C03637=1034.949,55.680,408.696,168.997,41.142,157.715
C03638=1034.955,55.929,408.679,168.999,41.142,157.715
C03639=1034.961,56.179,408.661,169.001,41.141,157.715
C03640=1034.968,56.428,408.644,169.004,41.140,157.715
C03641=1034.974,56.677,408.627,169.006,41.140,157.715
C03642=1034.980,56.927,408.610,169.008,41.139,157.715
C03643=1034.986,57.176,408.593,169.010,41.139,157.715
C03644=1034.993,57.425,408.576,169.012,41.139,157.715
C03645=1034.999,57.675,408.558,169.015,41.138,157.715
C03646=1035.006,57.924,408.541,169.017,41.138,157.715
C03647=1035.012,58.174,408.523,169.019,41.137,157.715
C03648=1035.018,58.423,408.505,169.021,41.136,157.715
C03649=1035.025,58.672,408.488,169.023,41.136,157.715
C03650=1035.031,58.921,408.470,169.026,41.136,157.715
C03651=1035.038,59.171,408.453,169.028,41.135,157.715
C03652=1035.044,59.420,408.436,169.030,41.135,157.715
C03653=1035.050,59.669,408.418,169.032,41.134,157.715
C03654=1035.056,59.918,408.401,169.034,41.134,157.715
C03655=1035.064,60.205,408.381,169.037,41.133,157.715
C03656=1035.071,60.491,408.361,169.039,41.132,157.715
C03657=1035.079,60.777,408.341,169.041,41.132,157.715
C03658=1035.086,61.063,408.321,169.044,41.131,157.715
C03659=1035.092,61.313,408.303,169.046,41.131,157.715
C03660=1035.099,61.561,408.286,169.048,41.130,157.715
C03661=1035.105,61.811,408.269,169.050,41.130,157.715
C03662=1035.112,62.061,408.251,169.052,41.129,157.715
C03663=1035.118,62.310,408.234,169.055,41.128,157.715
C03664=1035.125,62.558,408.216,169.057,41.128,157.715
C03665=1035.131,62.808,408.198,169.059,41.128,157.715
C03666=1035.138,63.057,408.181,169.061,41.127,157.715
C03667=1035.144,63.306,408.164,169.064,41.127,157.715
C03668=1035.150,63.556,408.146,169.066,41.126,157.715
C03669=1035.157,63.805,408.129,169.068,41.125,157.715
C03670=1035.163,64.055,408.111,169.070,41.125,157.715
C03671=1035.169,64.304,408.093,169.072,41.125,157.715
C03672=1035.176,64.553,408.075,169.074,41.124,157.715
C03673=1035.182,64.802,408.057,169.077,41.124,157.715
C03674=1035.188,65.052,408.039,169.079,41.123,157.715
C03675=1035.194,65.301,408.022,169.081,41.123,157.716
C03676=1035.201,65.551,408.004,169.083,41.122,157.715
C03677=1035.208,65.800,407.986,169.085,41.122,157.716
C03678=1035.213,66.049,407.969,169.088,41.122,157.716
C03679=1035.219,66.298,407.951,169.090,41.122,157.716
C03680=1035.226,66.548,407.933,169.092,41.121,157.716
C03681=1035.232,66.796,407.915,169.094,41.120,157.716
C03682=1035.238,67.046,407.897,169.096,41.120,157.716
C03683=1035.245,67.295,407.880,169.098,41.120,157.716
C03684=1035.251,67.544,407.861,169.101,41.119,157.716
C03685=1035.257,67.793,407.844,169.103,41.119,157.716
C03686=1035.263,68.043,407.826,169.105,41.118,157.716
C03687=1035.270,68.292,407.808,169.107,41.118,157.716
C03688=1035.276,68.542,407.790,169.109,41.117,157.716
C03689=1035.282,68.791,407.772,169.111,41.117,157.716
C03690=1035.289,69.040,407.754,169.114,41.117,157.716
C03691=1035.295,69.289,407.736,169.116,41.116,157.716
C03692=1035.301,69.539,407.718,169.118,41.116,157.716
C03693=1035.308,69.788,407.700,169.120,41.115,157.716
C03694=1035.313,70.037,407.682,169.122,41.115,157.716
C03695=1035.320,70.287,407.665,169.124,41.115,157.716
C03696=1035.327,70.536,407.646,169.127,41.114,157.716
C03697=1035.333,70.786,407.628,169.129,41.114,157.716
C03698=1035.338,71.034,407.610,169.131,41.113,157.716
C03699=1035.345,71.284,407.592,169.133,41.113,157.716
C03700=1035.351,71.533,407.573,169.135,41.113,157.716
C03701=1035.357,71.783,407.555,169.137,41.113,157.716
C03702=1035.364,72.031,407.537,169.140,41.112,157.717
C03703=1035.370,72.280,407.520,169.142,41.111,157.716
C03704=1035.376,72.530,407.502,169.144,41.111,157.717
C03705=1035.382,72.779,407.483,169.146,41.111,157.717
C03706=1035.388,73.029,407.465,169.148,41.111,157.717
C03707=1035.395,73.278,407.446,169.150,41.110,157.717
C03708=1035.400,73.527,407.429,169.152,41.110,157.717
C03709=1035.408,73.776,407.411,169.155,41.109,157.717
C03710=1035.414,74.025,407.392,169.157,41.109,157.717
C03711=1035.420,74.275,407.374,169.159,41.109,157.717
C03712=1035.427,74.524,407.356,169.161,41.108,157.717
C03713=1035.433,74.774,407.338,169.163,41.108,157.717
C03714=1035.439,75.022,407.319,169.165,41.107,157.717
C03715=1035.445,75.272,407.301,169.168,41.107,157.717
C03716=1035.451,75.521,407.283,169.170,41.107,157.717
C03717=1035.457,75.771,407.265,169.172,41.106,157.717
C03718=1035.464,76.020,407.247,169.174,41.106,157.717
C03719=1035.471,76.305,407.226,169.177,41.105,157.717
C03720=1035.479,76.591,407.205,169.179,41.105,157.717
C03721=1035.485,76.877,407.184,169.182,41.104,157.717
C03722=1035.493,77.163,407.163,169.184,41.104,157.717
C03723=1035.499,77.413,407.144,169.186,41.103,157.717
C03724=1035.506,77.662,407.126,169.188,41.103,157.717
C03725=1035.511,77.911,407.108,169.191,41.103,157.717
C03726=1035.518,78.160,407.089,169.193,41.103,157.717
C03727=1035.524,78.409,407.071,169.195,41.102,157.717
C03728=1035.530,78.659,407.053,169.197,41.102,157.717
C03729=1035.536,78.908,407.034,169.199,41.101,157.718
C03730=1035.542,79.157,407.015,169.201,41.101,157.718
C03731=1035.548,79.407,406.997,169.203,41.101,157.718
C03732=1035.555,79.656,406.978,169.206,41.100,157.718
C03733=1035.561,79.905,406.960,169.208,41.100,157.718
C03734=1035.567,80.154,406.941,169.210,41.100,157.718
C03735=1035.573,80.403,406.923,169.212,41.100,157.718
C03736=1035.579,80.653,406.904,169.214,41.099,157.718
C03737=1035.585,80.902,406.886,169.216,41.099,157.718
C03738=1035.592,81.151,406.867,169.218,41.098,157.718
C03739=1035.598,81.400,406.848,169.221,41.098,157.718
C03740=1035.604,81.650,406.830,169.223,41.098,157.718
C03741=1035.611,81.899,406.812,169.225,41.097,157.718
C03742=1035.616,82.149,406.792,169.227,41.097,157.718
C03743=1035.623,82.398,406.774,169.229,41.097,157.718
C03744=1035.629,82.646,406.756,169.231,41.096,157.718
C03745=1035.635,82.895,406.737,169.233,41.096,157.718
C03746=1035.641,83.145,406.719,169.236,41.096,157.718
C03747=1035.648,83.394,406.700,169.238,41.095,157.718
C03748=1035.653,83.643,406.681,169.240,41.095,157.719
C03749=1035.660,83.893,406.662,169.242,41.095,157.719
C03750=1035.666,84.142,406.644,169.244,41.095,157.719
C03751=1035.673,84.391,406.625,169.246,41.094,157.719
C03752=1035.679,84.640,406.606,169.249,41.093,157.719
C03753=1035.685,84.889,406.588,169.251,41.093,157.719
C03754=1035.691,85.139,406.569,169.253,41.093,157.719
C03755=1035.697,85.388,406.551,169.255,41.093,157.719
C03756=1035.704,85.637,406.532,169.257,41.092,157.719
C03757=1035.710,85.887,406.513,169.259,41.091,157.719
C03758=1035.717,86.136,406.495,169.262,41.091,157.719
C03759=1035.722,86.385,406.475,169.264,41.091,157.719
C03760=1035.729,86.634,406.457,169.266,41.091,157.719
C03761=1035.735,86.883,406.438,169.268,41.090,157.719
C03762=1035.742,87.132,406.420,169.270,41.090,157.719
C03763=1035.748,87.382,406.401,169.272,41.089,157.719
C03764=1035.754,87.631,406.382,169.275,41.089,157.719
C03765=1035.760,87.880,406.363,169.277,41.089,157.719
C03766=1035.766,88.129,406.344,169.279,41.088,157.719
C03767=1035.773,88.378,406.326,169.281,41.088,157.719
C03768=1035.779,88.627,406.307,169.283,41.087,157.719
C03769=1035.786,88.877,406.288,169.286,41.087,157.719
C03770=1035.791,89.126,406.269,169.288,41.087,157.719
C03771=1035.798,89.375,406.250,169.290,41.086,157.719
C03772=1035.805,89.625,406.231,169.292,41.086,157.720
C03773=1035.811,89.874,406.213,169.294,41.085,157.719
C03774=1035.817,90.124,406.194,169.296,41.085,157.720
C03775=1035.823,90.373,406.175,169.299,41.085,157.720
C03776=1035.829,90.622,406.156,169.301,41.084,157.720
C03777=1035.836,90.871,406.136,169.303,41.084,157.720
C03778=1035.842,91.120,406.117,169.305,41.084,157.720
C03779=1035.848,91.369,406.098,169.307,41.084,157.720
C03780=1035.854,91.619,406.079,169.309,41.084,157.720
C03781=1035.860,91.868,406.061,169.311,41.083,157.720
C03782=1035.867,92.117,406.042,169.314,41.083,157.720
C03783=1035.874,92.403,406.020,169.316,41.083,157.720
C03784=1035.880,92.688,405.998,169.319,41.082,157.720
C03785=1035.887,92.974,405.975,169.321,41.082,157.720
C03786=1035.894,93.260,405.954,169.324,41.082,157.720
C03787=1035.901,93.509,405.934,169.326,41.081,157.720
C03788=1035.907,93.758,405.915,169.328,41.081,157.721
C03789=1035.913,94.008,405.896,169.330,41.080,157.720
C03790=1035.919,94.257,405.877,169.332,41.080,157.720
C03791=1035.926,94.505,405.858,169.334,41.080,157.721
C03792=1035.931,94.755,405.839,169.336,41.080,157.721
C03793=1035.938,95.004,405.820,169.339,41.079,157.721
C03794=1035.944,95.254,405.800,169.341,41.079,157.721
C03795=1035.951,95.503,405.781,169.343,41.079,157.721
C03796=1035.956,95.752,405.762,169.345,41.079,157.721
C03797=1035.963,96.001,405.743,169.347,41.078,157.721
C03798=1035.969,96.251,405.724,169.349,41.078,157.721
C03799=1035.975,96.499,405.704,169.352,41.078,157.721
C03800=1035.981,96.749,405.685,169.354,41.077,157.721
C03801=1035.987,96.998,405.667,169.356,41.077,157.721
C03802=1035.994,97.247,405.646,169.358,41.076,157.721
C03803=1036.000,97.496,405.628,169.360,41.076,157.721
C03804=1036.006,97.746,405.608,169.363,41.076,157.721
C03805=1036.013,97.994,405.589,169.365,41.076,157.721
C03806=1036.018,98.244,405.570,169.367,41.075,157.721
C03807=1036.025,98.493,405.551,169.369,41.075,157.721
C03808=1036.032,98.742,405.531,169.371,41.075,157.722
C03809=1036.038,98.991,405.512,169.373,41.075,157.722
C03810=1036.044,99.240,405.492,169.376,41.074,157.722
C03811=1036.050,99.489,405.474,169.378,41.073,157.722
C03812=1036.056,99.739,405.454,169.380,41.073,157.722
C03813=1036.063,99.988,405.435,169.382,41.073,157.722
C03814=1036.069,100.237,405.415,169.384,41.073,157.722
C03815=1036.075,100.486,405.395,169.387,41.072,157.722
C03816=1036.081,100.735,405.377,169.389,41.072,157.722
C03817=1036.087,100.984,405.357,169.391,41.072,157.722
C03818=1036.093,101.234,405.338,169.393,41.071,157.722
C03819=1036.100,101.483,405.317,169.395,41.071,157.722
C03820=1036.106,101.732,405.299,169.397,41.071,157.722
C03821=1036.112,101.981,405.279,169.400,41.071,157.722
C03822=1036.118,102.231,405.259,169.402,41.070,157.722
C03823=1036.124,102.479,405.239,169.404,41.070,157.722
C03824=1036.130,102.729,405.220,169.406,41.070,157.722
C03825=1036.137,102.978,405.200,169.408,41.070,157.722
C03826=1036.143,103.227,405.180,169.411,41.069,157.723
C03827=1036.149,103.476,405.161,169.414,41.069,157.723
C03828=1036.155,103.725,405.141,169.416,41.069,157.723
C03829=1036.161,103.974,405.123,169.418,41.069,157.723
C03830=1036.168,104.224,405.102,169.420,41.068,157.723
C03831=1036.174,104.472,405.082,169.422,41.068,157.723
C03832=1036.179,104.722,405.063,169.424,41.068,157.723
C03833=1036.185,104.971,405.043,169.427,41.068,157.723
C03834=1036.192,105.221,405.024,169.429,41.067,157.723
C03835=1036.198,105.469,405.004,169.431,41.067,157.723
C03836=1036.204,105.718,404.984,169.433,41.067,157.723
C03837=1036.210,105.968,404.965,169.435,41.067,157.723
C03838=1036.217,106.217,404.945,169.438,41.066,157.723
C03839=1036.223,106.466,404.925,169.440,41.066,157.723
C03840=1036.229,106.715,404.906,169.442,41.066,157.723
C03841=1036.235,106.964,404.886,169.444,41.066,157.724
C03842=1036.242,107.213,404.866,169.446,41.065,157.724
C03843=1036.247,107.463,404.846,169.448,41.065,157.724
C03844=1036.254,107.711,404.827,169.451,41.065,157.724
C03845=1036.261,107.961,404.807,169.453,41.064,157.724
C03846=1036.267,108.210,404.787,169.455,41.064,157.724
C03847=1036.274,108.495,404.764,169.458,41.064,157.724
C03848=1036.281,108.781,404.742,169.460,41.064,157.724
C03849=1036.288,109.067,404.719,169.463,41.063,157.724
C03850=1036.295,109.353,404.696,169.465,41.063,157.724
C03851=1036.301,109.602,404.676,169.467,41.063,157.724
C03852=1036.308,109.852,404.657,169.470,41.062,157.724
C03853=1036.314,110.101,404.637,169.472,41.062,157.724
C03854=1036.320,110.349,404.617,169.474,41.062,157.724
C03855=1036.326,110.599,404.597,169.476,41.062,157.724
C03856=1036.332,110.848,404.577,169.478,41.061,157.725
C03857=1036.338,111.097,404.558,169.481,41.061,157.725
C03858=1036.345,111.347,404.538,169.483,41.061,157.725
C03859=1036.351,111.595,404.518,169.485,41.061,157.725
C03860=1036.357,111.844,404.498,169.487,41.060,157.725
C03861=1036.363,112.094,404.477,169.489,41.060,157.725
C03862=1036.369,112.343,404.457,169.492,41.060,157.725
C03863=1036.375,112.591,404.437,169.495,41.060,157.725
C03864=1036.382,112.841,404.417,169.497,41.059,157.725
C03865=1036.388,113.090,404.398,169.499,41.059,157.725
C03866=1036.394,113.340,404.377,169.501,41.059,157.725
C03867=1036.400,113.589,404.358,169.504,41.058,157.725
C03868=1036.406,113.837,404.338,169.506,41.058,157.725
C03869=1036.412,114.087,404.317,169.508,41.058,157.725
C03870=1036.418,114.336,404.297,169.510,41.058,157.726
C03871=1036.424,114.585,404.277,169.512,41.058,157.726
C03872=1036.430,114.834,404.257,169.515,41.058,157.726
C03873=1036.436,115.084,404.236,169.517,41.058,157.726
C03874=1036.442,115.332,404.216,169.519,41.057,157.726
C03875=1036.449,115.581,404.195,169.521,41.057,157.726
C03876=1036.455,115.830,404.175,169.523,41.057,157.726
C03877=1036.460,116.079,404.154,169.525,41.057,157.726
C03878=1036.467,116.329,404.134,169.528,41.057,157.726
C03879=1036.473,116.578,404.114,169.530,41.057,157.726
C03880=1036.479,116.826,404.094,169.532,41.056,157.726
C03881=1036.484,117.076,404.073,169.534,41.056,157.726
C03882=1036.490,117.325,404.053,169.536,41.057,157.727
C03883=1036.496,117.574,404.033,169.540,41.056,157.727
C03884=1036.503,117.823,404.013,169.542,41.056,157.727
C03885=1036.508,118.072,403.992,169.544,41.056,157.727
C03886=1036.515,118.321,403.971,169.546,41.055,157.727
C03887=1036.521,118.570,403.951,169.548,41.055,157.727
C03888=1036.527,118.819,403.931,169.551,41.055,157.727
C03889=1036.533,119.069,403.910,169.553,41.055,157.727
C03890=1036.539,119.318,403.891,169.555,41.055,157.727
C03891=1036.546,119.567,403.870,169.557,41.055,157.727
C03892=1036.552,119.815,403.850,169.559,41.055,157.727
C03893=1036.558,120.065,403.829,169.562,41.054,157.727
C03894=1036.564,120.314,403.809,169.564,41.054,157.728
C03895=1036.570,120.563,403.788,169.566,41.054,157.728
C03896=1036.576,120.813,403.768,169.568,41.053,157.728
C03897=1036.582,121.061,403.747,169.571,41.054,157.728
C03898=1036.589,121.310,403.727,169.573,41.054,157.728
C03899=1036.595,121.559,403.707,169.575,41.053,157.728
C03900=1036.600,121.809,403.686,169.577,41.053,157.728
C03901=1036.606,122.058,403.666,169.579,41.053,157.728
C03902=1036.613,122.307,403.645,169.582,41.052,157.728
C03903=1036.619,122.556,403.624,169.584,41.052,157.728
C03904=1036.625,122.805,403.604,169.586,41.052,157.728
C03905=1036.631,123.053,403.583,169.589,41.052,157.729
C03906=1036.638,123.303,403.563,169.592,41.052,157.729
C03907=1036.643,123.552,403.542,169.594,41.052,157.729
C03908=1036.650,123.802,403.522,169.596,41.052,157.729
C03909=1036.656,124.050,403.501,169.598,41.051,157.729
C03910=1036.662,124.300,403.481,169.601,41.051,157.729
C03911=1036.669,124.585,403.457,169.603,41.051,157.729
C03912=1036.676,124.870,403.433,169.606,41.050,157.729
C03913=1036.683,125.156,403.410,169.608,41.051,157.729
C03914=1036.690,125.443,403.386,169.611,41.050,157.729
C03915=1036.697,125.691,403.366,169.613,41.050,157.729
C03916=1036.703,125.940,403.345,169.615,41.050,157.729
C03917=1036.709,126.189,403.325,169.618,41.050,157.729
C03918=1036.715,126.438,403.304,169.620,41.049,157.730
C03919=1036.722,126.688,403.283,169.622,41.049,157.730
C03920=1036.728,126.936,403.263,169.625,41.049,157.730
C03921=1036.734,127.186,403.242,169.627,41.048,157.730
C03922=1036.740,127.435,403.222,169.629,41.048,157.730
C03923=1036.747,127.684,403.201,169.631,41.049,157.730
C03924=1036.752,127.933,403.180,169.634,41.048,157.730
C03925=1036.759,128.182,403.159,169.636,41.048,157.730
C03926=1036.766,128.431,403.139,169.638,41.048,157.730
C03927=1036.771,128.680,403.118,169.642,41.047,157.730
C03928=1036.778,128.929,403.097,169.644,41.047,157.730
C03929=1036.785,129.179,403.077,169.646,41.047,157.730
C03930=1036.790,129.427,403.056,169.648,41.047,157.730
C03931=1036.797,129.677,403.035,169.651,41.046,157.731
C03932=1036.803,129.925,403.015,169.653,41.046,157.731
C03933=1036.809,130.175,402.994,169.655,41.046,157.731
C03934=1036.816,130.424,402.973,169.658,41.046,157.731
C03935=1036.822,130.672,402.953,169.660,41.046,157.731
C03936=1036.828,130.922,402.931,169.662,41.046,157.731
C03937=1036.835,131.170,402.910,169.664,41.045,157.731
C03938=1036.840,131.420,402.889,169.667,41.045,157.731
C03939=1036.846,131.669,402.868,169.669,41.045,157.731
C03940=1036.852,131.918,402.848,169.671,41.045,157.731
C03941=1036.858,132.167,402.826,169.673,41.045,157.731
C03942=1036.865,132.416,402.805,169.676,41.045,157.732
C03943=1036.871,132.665,402.785,169.678,41.044,157.732
C03944=1036.877,132.914,402.763,169.680,41.045,157.732
C03945=1036.884,133.163,402.742,169.683,41.044,157.732
C03946=1036.889,133.412,402.721,169.685,41.044,157.732
C03947=1036.895,133.661,402.700,169.688,41.044,157.732
C03948=1036.901,133.909,402.679,169.690,41.044,157.732
C03949=1036.907,134.159,402.658,169.693,41.044,157.732
C03950=1036.913,134.408,402.637,169.695,41.044,157.732
C03951=1036.920,134.657,402.616,169.697,41.043,157.732
C03952=1036.926,134.906,402.594,169.700,41.044,157.733
C03953=1036.932,135.156,402.573,169.702,41.044,157.733
C03954=1036.938,135.404,402.553,169.704,41.043,157.733
C03955=1036.944,135.653,402.531,169.706,41.043,157.733
C03956=1036.951,135.902,402.510,169.709,41.043,157.733
C03957=1036.957,136.152,402.489,169.711,41.043,157.733
C03958=1036.962,136.400,402.468,169.713,41.043,157.733
C03959=1036.969,136.649,402.447,169.716,41.042,157.733
C03960=1036.976,136.898,402.425,169.719,41.043,157.733
C03961=1036.981,137.147,402.404,169.721,41.043,157.733
C03962=1036.987,137.397,402.383,169.724,41.042,157.734
C03963=1036.994,137.646,402.362,169.726,41.042,157.734
C03964=1036.999,137.894,402.341,169.728,41.042,157.734
C03965=1037.006,138.143,402.319,169.730,41.042,157.734
C03966=1037.012,138.393,402.297,169.733,41.042,157.734
C03967=1037.019,138.641,402.276,169.735,41.042,157.734
C03968=1037.024,138.891,402.256,169.737,41.042,157.734
C03969=1037.030,139.140,402.234,169.740,41.042,157.734
C03970=1037.036,139.389,402.212,169.742,41.041,157.734
C03971=1037.042,139.638,402.191,169.744,41.042,157.735
C03972=1037.049,139.886,402.170,169.747,41.041,157.735
C03973=1037.055,140.136,402.149,169.749,41.041,157.735
C03974=1037.061,140.385,402.127,169.752,41.042,157.735
C03975=1037.068,140.670,402.102,169.755,41.041,157.735
C03976=1037.075,140.955,402.078,169.758,41.042,157.735
C03977=1037.082,141.241,402.053,169.760,41.041,157.735
C03978=1037.088,141.526,402.028,169.763,41.041,157.735
C03979=1037.095,141.775,402.006,169.765,41.041,157.736
C03980=1037.101,142.025,401.985,169.767,41.041,157.736
C03981=1037.108,142.273,401.964,169.770,41.041,157.736
C03982=1037.113,142.522,401.942,169.772,41.041,157.736
C03983=1037.119,142.771,401.921,169.774,41.041,157.736
C03984=1037.125,143.020,401.899,169.777,41.041,157.736
C03985=1037.132,143.270,401.878,169.780,41.041,157.736
C03986=1037.137,143.518,401.856,169.782,41.041,157.736
C03987=1037.143,143.767,401.835,169.785,41.041,157.736
C03988=1037.150,144.016,401.813,169.787,41.041,157.737
C03989=1037.156,144.266,401.791,169.789,41.040,157.737
C03990=1037.162,144.515,401.770,169.792,41.041,157.737
C03991=1037.168,144.764,401.748,169.794,41.041,157.737
C03992=1037.174,145.012,401.726,169.797,41.040,157.737
C03993=1037.181,145.261,401.705,169.799,41.041,157.737
C03994=1037.187,145.510,401.683,169.801,41.040,157.737
C03995=1037.193,145.759,401.662,169.804,41.040,157.737
C03996=1037.199,146.008,401.640,169.806,41.040,157.737
C03997=1037.205,146.258,401.618,169.808,41.040,157.738
C03998=1037.211,146.506,401.597,169.812,41.040,157.738
C03999=1037.217,146.755,401.575,169.814,41.040,157.738
C04000=1037.224,147.004,401.553,169.816,41.040,157.738
C04001=1037.230,147.253,401.532,169.819,41.040,157.738
C04002=1037.236,147.502,401.510,169.821,41.040,157.738
C04003=1037.242,147.751,401.488,169.823,41.040,157.738
C04004=1037.249,148.000,401.466,169.826,41.040,157.738
C04005=1037.253,148.249,401.444,169.828,41.040,157.738
C04006=1037.260,148.498,401.422,169.831,41.040,157.739
C04007=1037.266,148.747,401.400,169.833,41.040,157.739
C04008=1037.272,148.996,401.378,169.836,41.040,157.739
C04009=1037.278,149.245,401.357,169.839,41.040,157.739
C04010=1037.285,149.494,401.335,169.841,41.040,157.739
C04011=1037.291,149.743,401.313,169.843,41.040,157.739
C04012=1037.296,149.993,401.291,169.846,41.040,157.739
C04013=1037.302,150.240,401.269,169.848,41.040,157.740
C04014=1037.308,150.490,401.247,169.850,41.040,157.740
C04015=1037.315,150.739,401.225,169.853,41.040,157.740
C04016=1037.321,150.987,401.203,169.855,41.040,157.740
C04017=1037.327,151.237,401.181,169.859,41.040,157.740
C04018=1037.333,151.485,401.158,169.861,41.040,157.740
C04019=1037.339,151.735,401.137,169.863,41.040,157.740
C04020=1037.345,151.984,401.115,169.866,41.040,157.740
C04021=1037.352,152.232,401.093,169.868,41.040,157.741
C04022=1037.358,152.482,401.071,169.870,41.040,157.741
C04023=1037.364,152.731,401.048,169.873,41.040,157.741
C04024=1037.370,152.980,401.027,169.875,41.040,157.741
C04025=1037.376,153.228,401.005,169.878,41.040,157.741
C04026=1037.382,153.477,400.983,169.880,41.040,157.741
C04027=1037.388,153.726,400.961,169.883,41.041,157.741
C04028=1037.394,153.975,400.938,169.886,41.040,157.742
C04029=1037.400,154.224,400.917,169.888,41.040,157.742
C04030=1037.406,154.473,400.894,169.891,41.040,157.742
C04031=1037.414,154.794,400.866,169.894,41.040,157.742
C04032=1037.422,155.115,400.836,169.897,41.040,157.742
C04033=1037.430,155.437,400.808,169.900,41.040,157.742
C04034=1037.438,155.758,400.780,169.903,41.041,157.743
C04035=1037.443,155.989,400.759,169.905,41.040,157.743
C04036=1037.449,156.219,400.738,169.909,41.041,157.743
C04037=1037.454,156.450,400.718,169.911,41.040,157.743
C04038=1037.460,156.682,400.697,169.913,41.041,157.743
C04039=1037.466,156.912,400.676,169.915,41.041,157.743
C04040=1037.471,157.143,400.656,169.917,41.041,157.743
C04041=1037.478,157.374,400.635,169.920,41.041,157.743
C04042=1037.483,157.605,400.614,169.922,41.041,157.744
C04043=1037.489,157.854,400.592,169.924,41.041,157.744
C04044=1037.495,158.103,400.569,169.928,41.041,157.744
C04045=1037.501,158.351,400.547,169.930,41.041,157.744
C04046=1037.507,158.601,400.525,169.933,41.041,157.744
C04047=1037.513,158.850,400.502,169.935,41.042,157.744
C04048=1037.520,159.098,400.480,169.938,41.041,157.744
C04049=1037.525,159.348,400.458,169.940,41.042,157.745
C04050=1037.532,159.596,400.436,169.942,41.041,157.745
C04051=1037.538,159.845,400.413,169.945,41.042,157.745
C04052=1037.545,160.094,400.390,169.947,41.041,157.745
C04053=1037.550,160.344,400.368,169.951,41.042,157.745
C04054=1037.556,160.593,400.345,169.953,41.042,157.745
C04055=1037.562,160.841,400.322,169.956,41.042,157.746
C04056=1037.568,161.090,400.299,169.958,41.043,157.746
C04057=1037.574,161.339,400.276,169.960,41.042,157.746
C04058=1037.580,161.588,400.254,169.963,41.043,157.746
C04059=1037.586,161.837,400.231,169.966,41.043,157.746
C04060=1037.592,162.086,400.208,169.969,41.043,157.747
C04061=1037.597,162.334,400.185,169.971,41.043,157.747
C04062=1037.603,162.584,400.163,169.973,41.044,157.747
C04063=1037.609,162.833,400.141,169.976,41.044,157.747
C04064=1037.615,163.081,400.118,169.978,41.044,157.747
C04065=1037.621,163.330,400.095,169.982,41.044,157.747
C04066=1037.626,163.579,400.072,169.984,41.044,157.747
C04067=1037.633,163.828,400.049,169.986,41.045,157.748
C04068=1037.639,164.077,400.027,169.989,41.045,157.748
C04069=1037.644,164.326,400.004,169.991,41.045,157.748
C04070=1037.650,164.575,399.981,169.994,41.046,157.748
C04071=1037.656,164.823,399.958,169.996,41.045,157.748
C04072=1037.662,165.072,399.935,170.000,41.046,157.749
C04073=1037.668,165.321,399.912,170.002,41.046,157.749
C04074=1037.674,165.571,399.889,170.005,41.046,157.749
C04075=1037.680,165.819,399.866,170.007,41.046,157.749
C04076=1037.686,166.068,399.842,170.009,41.046,157.749
C04077=1037.693,166.316,399.820,170.012,41.047,157.749
C04078=1037.698,166.565,399.797,170.015,41.047,157.750
C04079=1037.704,166.814,399.774,170.018,41.047,157.750
C04080=1037.710,167.063,399.751,170.020,41.047,157.750
C04081=1037.715,167.312,399.728,170.023,41.047,157.750
C04082=1037.723,167.561,399.706,170.025,41.048,157.750
C04083=1037.728,167.810,399.683,170.028,41.048,157.751
C04084=1037.734,168.059,399.660,170.031,41.048,157.751
C04085=1037.740,168.308,399.637,170.034,41.048,157.751
C04086=1037.746,168.556,399.613,170.036,41.048,157.751
C04087=1037.752,168.805,399.591,170.039,41.049,157.751
C04088=1037.759,169.054,399.567,170.041,41.049,157.751
C04089=1037.764,169.303,399.545,170.044,41.049,157.752
C04090=1037.770,169.552,399.522,170.046,41.049,157.752
C04091=1037.776,169.800,399.498,170.050,41.049,157.752
C04092=1037.782,170.049,399.475,170.052,41.050,157.752
C04093=1037.789,170.299,399.452,170.055,41.050,157.752
C04094=1037.795,170.547,399.429,170.057,41.051,157.753
C04095=1037.800,170.796,399.406,170.060,41.051,157.753
C04096=1037.806,171.045,399.383,170.062,41.051,157.753
C04097=1037.812,171.294,399.360,170.066,41.051,157.753
C04098=1037.818,171.543,399.336,170.068,41.051,157.753
C04099=1037.825,171.792,399.314,170.071,41.051,157.753
C04100=1037.831,172.040,399.290,170.073,41.052,157.754
C04101=1037.837,172.290,399.267,170.076,41.052,157.754
C04102=1037.843,172.538,399.244,170.078,41.052,157.754
C04103=1037.850,172.822,399.218,170.082,41.052,157.754
C04104=1037.857,173.108,399.191,170.085,41.052,157.754
C04105=1037.864,173.392,399.165,170.088,41.053,157.755
C04106=1037.871,173.677,399.138,170.091,41.053,157.755
C04107=1037.877,173.925,399.114,170.094,41.053,157.755
C04108=1037.883,174.175,399.091,170.097,41.054,157.755
C04109=1037.890,174.424,399.069,170.100,41.054,157.755
C04110=1037.896,174.672,399.045,170.102,41.054,157.755
C04111=1037.901,174.921,399.022,170.105,41.054,157.756
C04112=1037.908,175.170,398.998,170.107,41.054,157.756
C04113=1037.914,175.419,398.975,170.110,41.055,157.756
C04114=1037.920,175.667,398.952,170.114,41.055,157.756
C04115=1037.926,175.916,398.928,170.116,41.055,157.757
C04116=1037.933,176.165,398.906,170.119,41.055,157.757
C04117=1037.939,176.414,398.882,170.121,41.055,157.757
C04118=1037.945,176.663,398.859,170.124,41.056,157.757
C04119=1037.951,176.911,398.835,170.127,41.056,157.757
C04120=1037.957,177.161,398.812,170.130,41.056,157.757
C04121=1037.963,177.409,398.788,170.133,41.057,157.758
C04122=1037.969,177.658,398.765,170.135,41.057,157.758
C04123=1037.977,177.907,398.742,170.138,41.057,157.758
C04124=1037.982,178.156,398.719,170.141,41.057,157.758
C04125=1037.989,178.405,398.695,170.143,41.057,157.758
C04126=1037.995,178.653,398.672,170.147,41.057,157.759
C04127=1038.001,178.902,398.648,170.149,41.058,157.759
C04128=1038.007,179.151,398.625,170.152,41.058,157.759
C04129=1038.013,179.400,398.601,170.155,41.058,157.759
C04130=1038.019,179.649,398.578,170.157,41.059,157.759
C04131=1038.025,179.897,398.554,170.160,41.058,157.759
C04132=1038.033,180.146,398.531,170.164,41.059,157.760
C04133=1038.039,180.395,398.508,170.166,41.059,157.760
C04134=1038.045,180.644,398.484,170.169,41.059,157.760
C04135=1038.051,180.893,398.461,170.171,41.060,157.760
C04136=1038.058,181.142,398.437,170.174,41.060,157.761
C04137=1038.064,181.390,398.413,170.177,41.060,157.761
C04138=1038.070,181.640,398.390,170.180,41.061,157.761
C04139=1038.076,181.888,398.366,170.183,41.060,157.761
C04140=1038.083,182.137,398.342,170.186,41.061,157.761
C04141=1038.088,182.386,398.319,170.188,41.061,157.761
C04142=1038.096,182.635,398.296,170.191,41.061,157.762
C04143=1038.102,182.883,398.272,170.194,41.061,157.762
C04144=1038.108,183.132,398.249,170.197,41.062,157.762
C04145=1038.114,183.381,398.225,170.200,41.062,157.762
C04146=1038.120,183.630,398.201,170.203,41.062,157.763
C04147=1038.126,183.878,398.177,170.205,41.063,157.763
C04148=1038.133,184.127,398.153,170.208,41.063,157.763
C04149=1038.138,184.376,398.129,170.212,41.064,157.763
C04150=1038.144,184.624,398.105,170.214,41.064,157.763
C04151=1038.150,184.873,398.080,170.217,41.065,157.764
C04152=1038.156,185.122,398.057,170.219,41.065,157.764
C04153=1038.162,185.372,398.033,170.223,41.066,157.764
C04154=1038.168,185.620,398.009,170.226,41.066,157.764
C04155=1038.173,185.869,397.985,170.228,41.067,157.765
C04156=1038.180,186.117,397.961,170.231,41.067,157.765
C04157=1038.185,186.367,397.936,170.234,41.067,157.765
C04158=1038.191,186.615,397.913,170.237,41.068,157.765
C04159=1038.197,186.864,397.888,170.240,41.068,157.766
C04160=1038.203,187.113,397.864,170.242,41.069,157.766
C04161=1038.209,187.362,397.840,170.245,41.069,157.766
C04162=1038.215,187.610,397.816,170.249,41.070,157.766
C04163=1038.222,187.859,397.791,170.251,41.070,157.767
C04164=1038.228,188.107,397.767,170.254,41.071,157.767
C04165=1038.233,188.356,397.742,170.257,41.071,157.767
C04166=1038.240,188.605,397.719,170.260,41.072,157.767
C04167=1038.247,188.889,397.691,170.263,41.072,157.768
C04168=1038.253,189.173,397.664,170.266,41.073,157.768
C04169=1038.260,189.458,397.636,170.270,41.073,157.768
C04170=1038.267,189.742,397.608,170.273,41.074,157.768
C04171=1038.273,189.991,397.584,170.276,41.074,157.769
C04172=1038.279,190.240,397.559,170.279,41.075,157.769
C04173=1038.285,190.488,397.536,170.283,41.075,157.769
C04174=1038.291,190.737,397.510,170.285,41.076,157.770
C04175=1038.298,190.986,397.486,170.288,41.076,157.770
C04176=1038.303,191.234,397.462,170.291,41.077,157.770
C04177=1038.310,191.483,397.438,170.293,41.077,157.770
C04178=1038.315,191.732,397.414,170.297,41.078,157.771
C04179=1038.322,191.980,397.389,170.300,41.078,157.771
C04180=1038.328,192.230,397.364,170.302,41.078,157.771
C04181=1038.334,192.478,397.341,170.306,41.079,157.771
C04182=1038.340,192.727,397.316,170.309,41.080,157.772
C04183=1038.347,192.976,397.291,170.312,41.080,157.772
C04184=1038.352,193.224,397.267,170.314,41.081,157.772
C04185=1038.359,193.473,397.243,170.318,41.081,157.772
C04186=1038.365,193.722,397.218,170.321,41.081,157.773
C04187=1038.371,193.970,397.194,170.323,41.082,157.773
C04188=1038.377,194.219,397.170,170.326,41.083,157.773
C04189=1038.384,194.468,397.145,170.329,41.083,157.773
C04190=1038.389,194.716,397.121,170.333,41.083,157.774
C04191=1038.396,194.965,397.097,170.335,41.084,157.774
C04192=1038.402,195.214,397.071,170.338,41.085,157.774
C04193=1038.409,195.463,397.047,170.341,41.085,157.774
C04194=1038.414,195.712,397.023,170.345,41.086,157.775
C04195=1038.420,195.960,396.998,170.347,41.086,157.775
C04196=1038.427,196.209,396.974,170.350,41.087,157.775
C04197=1038.432,196.457,396.949,170.354,41.087,157.775
C04198=1038.439,196.706,396.925,170.357,41.087,157.776
C04199=1038.445,196.955,396.900,170.360,41.088,157.776
C04200=1038.452,197.204,396.875,170.362,41.089,157.776
C04201=1038.458,197.453,396.851,170.365,41.089,157.776
C04202=1038.464,197.701,396.826,170.369,41.090,157.777
C04203=1038.470,197.950,396.802,170.372,41.090,157.777
C04204=1038.476,198.199,396.776,170.375,41.090,157.777
C04205=1038.483,198.448,396.752,170.378,41.091,157.778
C04206=1038.488,198.696,396.727,170.381,41.092,157.778
C04207=1038.495,198.945,396.703,170.384,41.093,157.778
C04208=1038.501,199.193,396.678,170.387,41.093,157.778
C04209=1038.508,199.442,396.654,170.391,41.093,157.779
C04210=1038.514,199.691,396.628,170.393,41.094,157.779
C04211=1038.521,199.940,396.604,170.396,41.094,157.779
C04212=1038.526,200.188,396.579,170.399,41.095,157.779
C04213=1038.533,200.437,396.554,170.403,41.096,157.780
C04214=1038.539,200.686,396.530,170.406,41.096,157.780
C04215=1038.545,200.934,396.505,170.409,41.097,157.780
C04216=1038.552,201.183,396.479,170.412,41.098,157.781
C04217=1038.557,201.432,396.455,170.415,41.098,157.781
C04218=1038.564,201.681,396.429,170.418,41.099,157.781
C04219=1038.570,201.928,396.405,170.421,41.099,157.781
C04220=1038.576,202.178,396.380,170.425,41.100,157.782
C04221=1038.582,202.426,396.355,170.427,41.101,157.782
C04222=1038.588,202.675,396.330,170.430,41.101,157.782
C04223=1038.595,202.924,396.304,170.434,41.102,157.783
C04224=1038.601,203.172,396.279,170.437,41.102,157.783
C04225=1038.606,203.421,396.255,170.440,41.103,157.783
C04226=1038.612,203.670,396.230,170.443,41.104,157.784
C04227=1038.618,203.918,396.204,170.446,41.105,157.784
C04228=1038.625,204.167,396.179,170.449,41.105,157.784
C04229=1038.631,204.416,396.154,170.452,41.106,157.785
C04230=1038.638,204.664,396.129,170.456,41.107,157.785
C04231=1038.663,205.715,396.023,170.753,41.211,157.822
C04232=1038.672,206.029,395.989,170.757,41.212,157.823
C04233=1038.681,206.344,395.955,170.759,41.214,157.823
C04234=1038.690,206.658,395.923,170.762,41.216,157.824
C04235=1038.698,206.973,395.889,170.764,41.218,157.824
C04236=1038.704,207.221,395.863,170.767,41.220,157.825
C04237=1038.711,207.470,395.836,170.769,41.220,157.825
C04238=1038.718,207.718,395.809,170.772,41.222,157.826
C04239=1038.725,207.966,395.783,170.774,41.224,157.826
C04240=1038.731,208.215,395.756,170.776,41.225,157.826
C04241=1038.738,208.463,395.730,170.778,41.226,157.827
C04242=1038.745,208.712,395.704,170.781,41.228,157.827
C04243=1038.751,208.961,395.677,170.783,41.229,157.828
C04244=1038.758,209.209,395.651,170.786,41.231,157.828
C04245=1038.765,209.458,395.624,170.788,41.232,157.829
C04246=1038.771,209.707,395.597,170.790,41.233,157.829
C04247=1038.778,209.954,395.570,170.792,41.235,157.829
C04248=1038.785,210.203,395.544,170.795,41.237,157.830
C04249=1038.791,210.451,395.517,170.797,41.238,157.830
C04250=1038.798,210.700,395.491,170.800,41.239,157.831
C04251=1038.805,210.949,395.464,170.802,41.241,157.831
C04252=1038.811,211.197,395.437,170.803,41.242,157.831
C04253=1038.818,211.445,395.411,170.806,41.244,157.832
C04254=1038.825,211.695,395.384,170.809,41.245,157.832
C04255=1038.831,211.943,395.358,170.811,41.247,157.833
C04256=1038.838,212.191,395.330,170.813,41.248,157.833
C04257=1038.845,212.440,395.303,170.816,41.249,157.834
C04258=1038.851,212.688,395.277,170.819,41.251,157.834
C04259=1038.858,212.936,395.250,170.820,41.253,157.835
C04260=1038.864,213.185,395.223,170.822,41.254,157.835
C04261=1038.871,213.433,395.197,170.825,41.255,157.835
C04262=1038.878,213.682,395.169,170.827,41.257,157.836
C04263=1038.885,213.931,395.142,170.830,41.258,157.836
C04264=1038.890,214.179,395.116,170.832,41.260,157.837
C04265=1038.897,214.427,395.088,170.835,41.261,157.837
C04266=1038.904,214.676,395.062,170.836,41.263,157.838
C04267=1038.910,214.924,395.034,170.839,41.264,157.838
C04268=1038.917,215.173,395.008,170.841,41.266,157.838
C04269=1038.924,215.422,394.981,170.844,41.267,157.839
C04270=1038.931,215.670,394.954,170.846,41.268,157.839
C04271=1038.937,215.918,394.927,170.849,41.270,157.840
C04272=1038.944,216.166,394.900,170.851,41.271,157.840
C04273=1038.951,216.415,394.873,170.854,41.272,157.841
C04274=1038.958,216.664,394.845,170.856,41.274,157.841
C04275=1038.964,216.912,394.819,170.859,41.276,157.842
C04276=1038.970,217.161,394.792,170.860,41.277,157.842
C04277=1038.978,217.409,394.765,170.863,41.278,157.842
C04278=1038.984,217.658,394.738,170.865,41.280,157.843
C04279=1038.991,217.905,394.711,170.868,41.282,157.843
C04280=1038.997,218.155,394.684,170.870,41.283,157.844
C04281=1039.005,218.403,394.657,170.873,41.284,157.844
C04282=1039.012,218.651,394.629,170.875,41.286,157.845
C04283=1039.017,218.899,394.603,170.878,41.287,157.845
C04284=1039.025,219.148,394.576,170.880,41.288,157.845
C04285=1039.031,219.397,394.549,170.883,41.290,157.846
C04286=1039.038,219.645,394.521,170.885,41.291,157.846
C04287=1039.045,219.894,394.494,170.888,41.293,157.847
C04288=1039.053,220.213,394.459,170.890,41.295,157.847
C04289=1039.062,220.533,394.424,170.894,41.296,157.848
C04290=1039.070,220.854,394.389,170.896,41.299,157.848
C04291=1039.079,221.174,394.353,170.900,41.300,157.849
C04292=1039.085,221.421,394.327,170.903,41.302,157.849
C04293=1039.092,221.670,394.299,170.905,41.303,157.850
C04294=1039.099,221.918,394.271,170.908,41.305,157.850
C04295=1039.105,222.167,394.244,170.910,41.306,157.851
C04296=1039.112,222.416,394.217,170.913,41.307,157.851
C04297=1039.118,222.663,394.189,170.914,41.309,157.852
C04298=1039.125,222.912,394.163,170.917,41.311,157.852
C04299=1039.132,223.161,394.135,170.919,41.312,157.852
C04300=1039.138,223.409,394.107,170.922,41.313,157.853
C04301=1039.145,223.658,394.080,170.924,41.315,157.853
C04302=1039.152,223.906,394.052,170.927,41.317,157.854
C04303=1039.158,224.155,394.025,170.929,41.318,157.854
C04304=1039.164,224.403,393.997,170.932,41.319,157.855
C04305=1039.172,224.651,393.970,170.934,41.321,157.855
C04306=1039.178,224.899,393.943,170.937,41.322,157.856
C04307=1039.185,225.148,393.915,170.939,41.324,157.856
C04308=1039.192,225.396,393.887,170.942,41.325,157.856
C04309=1039.198,225.645,393.859,170.944,41.327,157.857
C04310=1039.205,225.894,393.832,170.947,41.328,157.857
C04311=1039.211,226.142,393.805,170.949,41.330,157.858
C04312=1039.219,226.390,393.777,170.952,41.331,157.858
C04313=1039.225,226.638,393.750,170.954,41.332,157.859
C04314=1039.232,226.886,393.722,170.957,41.334,157.859
C04315=1039.238,227.135,393.695,170.960,41.335,157.860
C04316=1039.245,227.383,393.667,170.963,41.336,157.860
C04317=1039.252,227.632,393.639,170.965,41.338,157.861
C04318=1039.258,227.880,393.611,170.968,41.340,157.861
C04319=1039.265,228.129,393.584,170.970,41.341,157.861
C04320=1039.272,228.377,393.557,170.972,41.342,157.862
C04321=1039.278,228.626,393.528,170.975,41.344,157.862
C04322=1039.285,228.874,393.501,170.978,41.345,157.863
C04323=1039.292,229.122,393.473,170.980,41.347,157.863
C04324=1039.298,229.371,393.445,170.982,41.348,157.864
C04325=1039.305,229.619,393.417,170.985,41.350,157.864
C04326=1039.312,229.868,393.390,170.988,41.351,157.865
C04327=1039.319,230.116,393.362,170.990,41.353,157.865
C04328=1039.325,230.365,393.334,170.993,41.354,157.866
C04329=1039.332,230.613,393.306,170.995,41.356,157.866
C04330=1039.339,230.861,393.278,170.998,41.357,157.866
C04331=1039.346,231.109,393.250,171.000,41.359,157.867
C04332=1039.351,231.358,393.222,171.003,41.360,157.867
C04333=1039.358,231.607,393.194,171.005,41.362,157.868
C04334=1039.365,231.855,393.166,171.008,41.363,157.868
C04335=1039.372,232.103,393.139,171.011,41.365,157.869
C04336=1039.379,232.351,393.110,171.014,41.366,157.869
C04337=1039.385,232.599,393.083,171.016,41.367,157.870
C04338=1039.391,232.848,393.055,171.019,41.369,157.870
C04339=1039.397,233.096,393.027,171.021,41.371,157.871
C04340=1039.404,233.344,392.998,171.024,41.372,157.871
C04341=1039.411,233.592,392.971,171.026,41.374,157.872
C04342=1039.417,233.842,392.942,171.029,41.375,157.872
C04343=1039.424,234.090,392.914,171.031,41.377,157.872
C04344=1039.433,234.402,392.879,171.035,41.378,157.873
C04345=1039.441,234.715,392.844,171.038,41.381,157.874
C04346=1039.449,235.027,392.808,171.041,41.382,157.874
C04347=1039.458,235.339,392.772,171.045,41.384,157.875
C04348=1039.464,235.588,392.745,171.048,41.386,157.875
C04349=1039.470,235.837,392.716,171.050,41.387,157.876
C04350=1039.477,236.084,392.688,171.053,41.389,157.876
C04351=1039.484,236.333,392.660,171.055,41.390,157.877
C04352=1039.491,236.581,392.632,171.058,41.392,157.877
C04353=1039.497,236.829,392.603,171.061,41.393,157.878
C04354=1039.504,237.079,392.575,171.064,41.395,157.878
C04355=1039.511,237.326,392.547,171.066,41.396,157.879
C04356=1039.518,237.575,392.519,171.069,41.398,157.879
C04357=1039.524,237.823,392.490,171.071,41.399,157.879
C04358=1039.531,238.071,392.462,171.074,41.400,157.880
C04359=1039.538,238.319,392.434,171.076,41.402,157.880
C04360=1039.544,238.568,392.406,171.080,41.403,157.881
C04361=1039.551,238.816,392.377,171.082,41.405,157.881
C04362=1039.558,239.065,392.349,171.085,41.407,157.882
C04363=1039.564,239.313,392.320,171.087,41.408,157.882
C04364=1039.571,239.561,392.292,171.090,41.410,157.883
C04365=1039.578,239.809,392.264,171.093,41.411,157.883
C04366=1039.584,240.058,392.236,171.096,41.412,157.884
C04367=1039.591,240.306,392.207,171.098,41.414,157.884
C04368=1039.598,240.554,392.179,171.101,41.415,157.885
C04369=1039.604,240.803,392.150,171.104,41.417,157.885
C04370=1039.611,241.051,392.122,171.106,41.419,157.886
C04371=1039.617,241.299,392.093,171.110,41.420,157.886
C04372=1039.624,241.548,392.065,171.112,41.422,157.887
C04373=1039.630,241.796,392.036,171.115,41.423,157.887
C04374=1039.637,242.044,392.007,171.117,41.425,157.888
C04375=1039.643,242.292,391.979,171.120,41.426,157.888
C04376=1039.650,242.541,391.950,171.122,41.428,157.888
C04377=1039.657,242.789,391.921,171.126,41.429,157.889
C04378=1039.663,243.037,391.892,171.129,41.431,157.889
C04379=1039.670,243.285,391.864,171.131,41.433,157.890
C04380=1039.676,243.534,391.835,171.134,41.434,157.890
C04381=1039.683,243.782,391.806,171.136,41.436,157.891
C04382=1039.690,244.030,391.777,171.140,41.437,157.891
C04383=1039.696,244.279,391.749,171.142,41.439,157.892
C04384=1039.703,244.527,391.721,171.145,41.440,157.892
C04385=1039.709,244.775,391.692,171.147,41.442,157.893
C04386=1039.716,245.024,391.662,171.151,41.443,157.893
C04387=1039.723,245.272,391.634,171.153,41.445,157.894
C04388=1039.729,245.520,391.605,171.156,41.447,157.894
C04389=1039.736,245.768,391.576,171.159,41.448,157.895
C04390=1039.742,246.016,391.547,171.161,41.450,157.895
C04391=1039.749,246.265,391.517,171.165,41.451,157.896
C04392=1039.756,246.513,391.489,171.167,41.453,157.896
C04393=1039.762,246.761,391.460,171.170,41.454,157.897
C04394=1039.768,247.009,391.431,171.172,41.456,157.897
C04395=1039.775,247.257,391.402,171.175,41.458,157.898
C04396=1039.781,247.506,391.372,171.179,41.460,157.898
C04397=1039.788,247.754,391.343,171.181,41.461,157.899
C04398=1039.794,248.002,391.314,171.184,41.463,157.899
C04399=1039.801,248.250,391.286,171.186,41.464,157.900
C04400=1039.809,248.558,391.250,171.190,41.466,157.901
C04401=1039.817,248.864,391.214,171.194,41.468,157.901
C04402=1039.825,249.170,391.178,171.197,41.470,157.902
C04403=1039.834,249.477,391.142,171.201,41.472,157.902
C04404=1039.840,249.725,391.113,171.204,41.474,157.903
C04405=1039.846,249.974,391.084,171.206,41.475,157.903
C04406=1039.853,250.222,391.054,171.209,41.477,157.904
C04407=1039.859,250.471,391.025,171.212,41.478,157.904
C04408=1039.866,250.718,390.995,171.215,41.480,157.905
C04409=1039.872,250.966,390.966,171.218,41.482,157.905
C04410=1039.879,251.215,390.937,171.221,41.483,157.906
C04411=1039.886,251.463,390.909,171.224,41.485,157.906
C04412=1039.892,251.711,390.880,171.226,41.487,157.907
C04413=1039.899,251.960,390.850,171.229,41.488,157.907
C04414=1039.906,252.207,390.820,171.232,41.490,157.908
C04415=1039.912,252.456,390.791,171.235,41.491,157.908
C04416=1039.919,252.704,390.762,171.237,41.493,157.909
C04417=1039.925,252.952,390.733,171.241,41.494,157.909
C04418=1039.932,253.201,390.703,171.244,41.496,157.910
C04419=1039.939,253.448,390.674,171.246,41.498,157.911
C04420=1039.945,253.697,390.645,171.250,41.499,157.911
C04421=1039.952,253.945,390.615,171.252,41.501,157.912
C04422=1039.959,254.193,390.586,171.255,41.503,157.912
C04423=1039.966,254.442,390.557,171.259,41.504,157.913
C04424=1039.972,254.689,390.527,171.261,41.506,157.913
C04425=1039.979,254.938,390.498,171.264,41.507,157.914
C04426=1039.985,255.186,390.468,171.267,41.509,157.914
C04427=1039.992,255.434,390.439,171.270,41.510,157.915
C04428=1039.999,255.683,390.409,171.273,41.512,157.915
C04429=1040.006,255.930,390.381,171.276,41.513,157.916
C04430=1040.013,256.179,390.351,171.279,41.515,157.916
C04431=1040.019,256.427,390.322,171.282,41.517,157.917
C04432=1040.026,256.675,390.292,171.285,41.518,157.917
C04433=1040.032,256.923,390.263,171.287,41.520,157.918
C04434=1040.040,257.171,390.232,171.291,41.521,157.918
C04435=1040.046,257.419,390.203,171.293,41.523,157.919
C04436=1040.053,257.668,390.174,171.297,41.524,157.919
C04437=1040.059,257.916,390.144,171.300,41.526,157.920
C04438=1040.066,258.165,390.115,171.302,41.528,157.920
C04439=1040.073,258.412,390.085,171.306,41.530,157.921
C04440=1040.080,258.661,390.056,171.308,41.531,157.921
C04441=1040.087,258.908,390.026,171.312,41.533,157.922
C04442=1040.094,259.157,389.997,171.315,41.534,157.922
C04443=1040.100,259.404,389.967,171.318,41.536,157.923
C04444=1040.107,259.653,389.937,171.321,41.537,157.923
C04445=1040.114,259.902,389.908,171.323,41.539,157.924
C04446=1040.121,260.149,389.878,171.327,41.540,157.924
C04447=1040.128,260.398,389.849,171.329,41.542,157.925
C04448=1040.134,260.645,389.819,171.333,41.544,157.925
C04449=1040.141,260.894,389.789,171.336,41.545,157.926
C04450=1040.148,261.142,389.759,171.339,41.547,157.926
C04451=1040.155,261.390,389.730,171.342,41.548,157.927
C04452=1040.162,261.638,389.699,171.345,41.550,157.928
C04453=1040.168,261.886,389.670,171.348,41.551,157.928
C04454=1040.175,262.135,389.640,171.350,41.553,157.928
C04455=1040.182,262.382,389.611,171.354,41.555,157.929
C04456=1040.190,262.688,389.574,171.358,41.557,157.930
C04457=1040.198,262.994,389.537,171.362,41.559,157.930
C04458=1040.206,263.298,389.500,171.365,41.561,157.931
C04459=1040.215,263.603,389.463,171.369,41.563,157.932
C04460=1040.221,263.852,389.433,171.372,41.565,157.932
C04461=1040.228,264.099,389.403,171.375,41.566,157.933
C04462=1040.235,264.348,389.373,171.378,41.568,157.933
C04463=1040.241,264.596,389.342,171.382,41.570,157.934
C04464=1040.248,264.844,389.312,171.384,41.571,157.934
C04465=1040.255,265.092,389.282,171.388,41.573,157.935
C04466=1040.261,265.340,389.252,171.390,41.575,157.936
C04467=1040.268,265.588,389.222,171.394,41.576,157.936
C04468=1040.275,265.836,389.192,171.397,41.579,157.937
C04469=1040.281,266.085,389.162,171.400,41.580,157.937
C04470=1040.288,266.333,389.132,171.403,41.582,157.938
C04471=1040.295,266.581,389.102,171.407,41.584,157.938
C04472=1040.301,266.829,389.071,171.409,41.585,157.939
C04473=1040.308,267.077,389.041,171.413,41.587,157.939
C04474=1040.315,267.325,389.010,171.416,41.589,157.940
C04475=1040.321,267.572,388.980,171.419,41.590,157.941
C04476=1040.328,267.821,388.950,171.422,41.592,157.941
C04477=1040.335,268.069,388.919,171.425,41.594,157.942
C04478=1040.341,268.317,388.889,171.428,41.595,157.942
C04479=1040.348,268.565,388.859,171.432,41.597,157.943
C04480=1040.355,268.813,388.829,171.434,41.599,157.943
C04481=1040.361,269.061,388.799,171.438,41.600,157.944
C04482=1040.368,269.309,388.767,171.441,41.603,157.945
C04483=1040.375,269.557,388.737,171.444,41.604,157.945
C04484=1040.382,269.806,388.707,171.447,41.606,157.946
C04485=1040.388,270.053,388.677,171.451,41.608,157.946
C04486=1040.395,270.302,388.646,171.453,41.609,157.947
C04487=1040.402,270.549,388.615,171.457,41.611,157.947
C04488=1040.409,270.798,388.584,171.460,41.613,157.948
C04489=1040.415,271.045,388.555,171.463,41.615,157.949
C04490=1040.421,271.294,388.524,171.467,41.616,157.949
C04491=1040.429,271.541,388.493,171.469,41.618,157.950
C04492=1040.435,271.790,388.462,171.473,41.620,157.950
C04493=1040.441,272.038,388.432,171.476,41.621,157.951
C04494=1040.449,272.285,388.401,171.479,41.623,157.951
C04495=1040.455,272.534,388.371,171.482,41.625,157.952
C04496=1040.461,272.782,388.340,171.486,41.627,157.953
C04497=1040.468,273.029,388.309,171.489,41.628,157.953
C04498=1040.475,273.278,388.279,171.492,41.631,157.954
C04499=1040.481,273.526,388.247,171.496,41.632,157.954
C04500=1040.489,273.774,388.217,171.498,41.634,157.955
C04501=1040.495,274.022,388.186,171.502,41.636,157.955
C04502=1040.501,274.270,388.155,171.505,41.638,157.956
C04503=1040.508,274.518,388.125,171.508,41.639,157.957
C04504=1040.515,274.766,388.094,171.512,41.641,157.957
C04505=1040.522,275.014,388.062,171.515,41.643,157.958
C04506=1040.529,275.262,388.032,171.518,41.645,157.958
C04507=1040.535,275.509,388.001,171.521,41.647,157.959
C04508=1040.541,275.758,387.970,171.525,41.648,157.960
C04509=1040.548,276.006,387.939,171.528,41.650,157.960
C04510=1040.555,276.254,387.909,171.531,41.652,157.961
C04511=1040.562,276.502,387.877,171.535,41.654,157.961
C04512=1040.570,276.812,387.838,171.538,41.656,157.962
C04513=1040.579,277.121,387.800,171.543,41.658,157.963
C04514=1040.587,277.431,387.761,171.547,41.660,157.964
C04515=1040.595,277.741,387.723,171.551,41.663,157.964
C04516=1040.603,277.989,387.692,171.555,41.664,157.965
C04517=1040.609,278.237,387.660,171.557,41.667,157.965
C04518=1040.616,278.485,387.630,171.561,41.668,157.966
C04519=1040.622,278.733,387.599,171.565,41.670,157.967
C04520=1040.629,278.980,387.567,171.568,41.672,157.967
C04521=1040.635,279.228,387.536,171.571,41.674,157.968
C04522=1040.642,279.476,387.504,171.575,41.676,157.968
C04523=1040.649,279.725,387.474,171.578,41.678,157.969
C04524=1040.655,279.973,387.442,171.581,41.680,157.970
C04525=1040.662,280.221,387.411,171.585,41.681,157.970
C04526=1040.669,280.469,387.379,171.588,41.683,157.971
C04527=1040.675,280.716,387.348,171.591,41.685,157.972
C04528=1040.683,280.964,387.317,171.595,41.687,157.972
C04529=1040.690,281.212,387.286,171.598,41.689,157.973
C04530=1040.696,281.460,387.254,171.602,41.691,157.973
C04531=1040.703,281.708,387.223,171.605,41.693,157.974
C04532=1040.710,281.956,387.192,171.608,41.695,157.975
C04533=1040.716,282.204,387.161,171.612,41.697,157.975
C04534=1040.722,282.451,387.130,171.615,41.699,157.976
C04535=1040.729,282.699,387.098,171.618,41.700,157.976
C04536=1040.736,282.947,387.067,171.622,41.702,157.977
C04537=1040.743,283.195,387.035,171.625,41.704,157.978
C04538=1040.750,283.444,387.003,171.629,41.706,157.978
C04539=1040.757,283.692,386.972,171.632,41.708,157.979
C04540=1040.764,283.939,386.940,171.636,41.710,157.980
C04541=1040.770,284.187,386.908,171.639,41.712,157.980
C04542=1040.776,284.435,386.876,171.642,41.714,157.981
C04543=1040.783,284.683,386.845,171.646,41.715,157.981
C04544=1040.790,284.931,386.814,171.649,41.717,157.982
C04545=1040.797,285.179,386.782,171.653,41.719,157.983
C04546=1040.803,285.427,386.751,171.656,41.721,157.983
C04547=1040.810,285.674,386.719,171.660,41.723,157.984
C04548=1040.817,285.922,386.688,171.663,41.725,157.985
C04549=1040.824,286.170,386.656,171.667,41.727,157.985
C04550=1040.830,286.418,386.624,171.671,41.729,157.986
C04551=1040.837,286.665,386.593,171.674,41.731,157.987
C04552=1040.844,286.914,386.561,171.677,41.733,157.987
C04553=1040.851,287.162,386.530,171.681,41.734,157.988
C04554=1040.858,287.409,386.497,171.685,41.736,157.989
C04555=1040.865,287.657,386.466,171.687,41.739,157.989
C04556=1040.871,287.905,386.434,171.691,41.741,157.990
C04557=1040.878,288.153,386.402,171.695,41.743,157.991
C04558=1040.885,288.401,386.370,171.699,41.745,157.991
C04559=1040.891,288.648,386.339,171.702,41.747,157.992
C04560=1040.899,288.896,386.306,171.705,41.749,157.992
C04561=1040.905,289.145,386.274,171.709,41.751,157.993
C04562=1040.912,289.392,386.242,171.713,41.753,157.994
C04563=1040.919,289.640,386.211,171.717,41.755,157.995
C04564=1040.926,289.888,386.179,171.719,41.756,157.995
C04565=1040.932,290.135,386.147,171.723,41.758,157.996
C04566=1040.939,290.384,386.115,171.727,41.760,157.996
C04567=1040.946,290.631,386.083,171.730,41.762,157.997
C04568=1040.955,290.952,386.041,171.736,41.765,157.998
C04569=1040.963,291.275,385.999,171.740,41.768,157.999
C04570=1040.972,291.596,385.958,171.745,41.770,158.000
C04571=1040.981,291.918,385.915,171.749,41.773,158.001
C04572=1040.988,292.166,385.884,171.752,41.775,158.001
C04573=1040.995,292.413,385.852,171.756,41.777,158.002
C04574=1041.001,292.661,385.820,171.760,41.779,158.003
C04575=1041.008,292.909,385.788,171.764,41.781,158.003
C04576=1041.015,293.157,385.755,171.767,41.783,158.004
C04577=1041.021,293.405,385.723,171.771,41.785,158.005
C04578=1041.028,293.652,385.691,171.775,41.787,158.005
C04579=1041.035,293.900,385.658,171.778,41.789,158.006
C04580=1041.042,294.148,385.626,171.782,41.792,158.007
C04581=1041.049,294.396,385.594,171.785,41.794,158.007
C04582=1041.055,294.643,385.562,171.789,41.796,158.008
C04583=1041.063,294.891,385.529,171.793,41.798,158.009
C04584=1041.069,295.139,385.496,171.797,41.800,158.009
C04585=1041.076,295.387,385.465,171.800,41.802,158.010
C04586=1041.083,295.635,385.432,171.804,41.804,158.011
C04587=1041.089,295.883,385.399,171.807,41.807,158.012
C04588=1041.096,296.130,385.367,171.811,41.809,158.012
C04589=1041.103,296.377,385.334,171.815,41.811,158.013
C04590=1041.109,296.626,385.301,171.818,41.813,158.014
C04591=1041.116,296.873,385.268,171.822,41.815,158.014
C04592=1041.123,297.121,385.236,171.826,41.817,158.015
C04593=1041.129,297.368,385.203,171.830,41.819,158.016
C04594=1041.136,297.616,385.170,171.834,41.822,158.017
C04595=1041.142,297.864,385.138,171.837,41.824,158.017
C04596=1041.149,298.112,385.105,171.841,41.826,158.018
C04597=1041.156,298.360,385.072,171.844,41.828,158.019
C04598=1041.162,298.607,385.040,171.848,41.830,158.019
C04599=1041.169,298.855,385.007,171.852,41.832,158.020
C04600=1041.176,299.103,384.974,171.856,41.834,158.021
C04601=1041.183,299.350,384.942,171.860,41.837,158.022
C04602=1041.189,299.597,384.908,171.864,41.839,158.022
C04603=1041.196,299.846,384.875,171.867,41.841,158.023
C04604=1041.202,300.093,384.842,171.871,41.844,158.024
C04605=1041.209,300.342,384.809,171.875,41.845,158.024
C04606=1041.216,300.589,384.777,171.879,41.847,158.025
C04607=1041.223,300.836,384.743,171.883,41.850,158.026
C04608=1041.230,301.084,384.710,171.886,41.852,158.027
C04609=1041.236,301.332,384.678,171.890,41.855,158.027
C04610=1041.243,301.580,384.645,171.893,41.857,158.028
C04611=1041.250,301.827,384.612,171.897,41.859,158.029
C04612=1041.257,302.075,384.579,171.901,41.861,158.030
C04613=1041.264,302.322,384.546,171.905,41.863,158.030
C04614=1041.270,302.571,384.513,171.909,41.866,158.031
C04615=1041.277,302.818,384.479,171.913,41.868,158.032
C04616=1041.285,303.066,384.447,171.916,41.870,158.032
C04617=1041.291,303.313,384.414,171.920,41.872,158.033
C04618=1041.298,303.561,384.380,171.924,41.874,158.034
C04619=1041.305,303.809,384.347,171.928,41.877,158.035
C04620=1041.312,304.056,384.314,171.932,41.879,158.035
C04621=1041.318,304.304,384.281,171.936,41.882,158.036
C04622=1041.326,304.552,384.248,171.940,41.884,158.037
C04623=1041.332,304.799,384.215,171.944,41.886,158.038
C04624=1041.341,305.137,384.169,171.950,41.889,158.039
C04625=1041.351,305.476,384.124,171.955,41.892,158.040
C04626=1041.360,305.814,384.079,171.960,41.895,158.041
C04627=1041.370,306.152,384.034,171.965,41.898,158.042
C04628=1041.377,306.400,384.000,171.969,41.901,158.043
C04629=1041.384,306.647,383.967,171.973,41.903,158.043
C04630=1041.391,306.895,383.934,171.977,41.905,158.044
C04631=1041.398,307.143,383.900,171.981,41.907,158.045
C04632=1041.404,307.390,383.867,171.985,41.910,158.046
C04633=1041.412,307.637,383.834,171.990,41.912,158.046
C04634=1041.419,307.885,383.800,171.993,41.914,158.047
C04635=1041.426,308.133,383.767,171.997,41.916,158.048
C04636=1041.433,308.380,383.733,172.001,41.919,158.049
C04637=1041.440,308.628,383.700,172.005,41.921,158.049
C04638=1041.446,308.876,383.667,172.009,41.923,158.050
C04639=1041.453,309.123,383.633,172.013,41.926,158.051
C04640=1041.461,309.371,383.600,172.017,41.928,158.052
C04641=1041.469,309.618,383.566,172.021,41.930,158.053
C04642=1041.475,309.866,383.533,172.026,41.932,158.053
C04643=1041.482,310.114,383.499,172.030,41.935,158.054
C04644=1041.489,310.361,383.466,172.033,41.937,158.055
C04645=1041.496,310.609,383.432,172.037,41.939,158.056
C04646=1041.503,310.857,383.399,172.041,41.942,158.056
C04647=1041.510,311.104,383.365,172.045,41.944,158.057
C04648=1041.518,311.352,383.332,172.049,41.946,158.058
C04649=1041.525,311.599,383.298,172.054,41.949,158.059
C04650=1041.532,311.847,383.264,172.058,41.951,158.060
C04651=1041.539,312.094,383.231,172.062,41.953,158.060
C04652=1041.546,312.342,383.197,172.066,41.956,158.061
C04653=1041.553,312.590,383.163,172.070,41.958,158.062
C04654=1041.560,312.837,383.129,172.074,41.961,158.063
C04655=1041.566,313.084,383.095,172.079,41.963,158.064
C04656=1041.573,313.332,383.061,172.083,41.966,158.065
C04657=1041.580,313.580,383.027,172.086,41.968,158.065
C04658=1041.587,313.827,382.992,172.090,41.971,158.066
C04659=1041.593,314.074,382.958,172.094,41.973,158.067
C04660=1041.600,314.322,382.924,172.098,41.976,158.068
C04661=1041.607,314.570,382.890,172.102,41.978,158.069
C04662=1041.614,314.818,382.856,172.107,41.981,158.069
C04663=1041.621,315.065,382.821,172.111,41.983,158.070
C04664=1041.627,315.312,382.787,172.115,41.986,158.071
C04665=1041.634,315.560,382.753,172.119,41.988,158.072
C04666=1041.641,315.808,382.719,172.123,41.991,158.073
C04667=1041.648,316.055,382.684,172.127,41.993,158.074
C04668=1041.655,316.303,382.651,172.132,41.996,158.074
C04669=1041.662,316.551,382.616,172.136,41.998,158.075
C04670=1041.669,316.798,382.582,172.140,42.001,158.076
C04671=1041.675,317.045,382.548,172.144,42.004,158.077
C04672=1041.682,317.293,382.514,172.148,42.007,158.078
C04673=1041.689,317.540,382.479,172.153,42.009,158.079
C04674=1041.696,317.788,382.445,172.157,42.012,158.080
C04675=1041.703,318.035,382.410,172.161,42.014,158.081
C04676=1041.710,318.283,382.376,172.165,42.017,158.081
C04677=1041.717,318.530,382.341,172.170,42.019,158.082
C04678=1041.724,318.778,382.307,172.174,42.022,158.083
C04679=1041.731,319.025,382.272,172.178,42.024,158.084
C04680=1041.741,319.368,382.224,172.185,42.028,158.085
C04681=1041.751,319.711,382.176,172.190,42.032,158.086
C04682=1041.760,320.054,382.129,172.197,42.035,158.088
C04683=1041.769,320.396,382.081,172.202,42.039,158.089
C04684=1041.777,320.644,382.045,172.206,42.041,158.090
C04685=1041.784,320.892,382.012,172.211,42.044,158.090
C04686=1041.791,321.139,381.976,172.215,42.046,158.091
C04687=1041.798,321.387,381.943,172.219,42.049,158.092
C04688=1041.805,321.634,381.907,172.224,42.052,158.093
C04689=1041.812,321.881,381.873,172.228,42.054,158.094
C04690=1041.819,322.129,381.838,172.232,42.057,158.095
C04691=1041.826,322.377,381.804,172.237,42.060,158.096
C04692=1041.833,322.624,381.769,172.241,42.062,158.097
C04693=1041.841,322.871,381.734,172.245,42.065,158.098
C04694=1041.848,323.120,381.699,172.250,42.067,158.098
C04695=1041.855,323.367,381.665,172.255,42.071,158.099
C04696=1041.862,323.614,381.630,172.259,42.073,158.100
C04697=1041.869,323.861,381.595,172.264,42.075,158.101
C04698=1041.876,324.108,381.560,172.268,42.078,158.102
C04699=1041.883,324.356,381.525,172.272,42.081,158.103
C04700=1041.891,324.604,381.491,172.277,42.084,158.104
C04701=1041.897,324.852,381.456,172.281,42.086,158.105
C04702=1041.905,325.099,381.421,172.285,42.089,158.106
C04703=1041.912,325.346,381.386,172.290,42.092,158.107
C04704=1041.920,325.594,381.351,172.294,42.095,158.108
C04705=1041.927,325.841,381.316,172.299,42.097,158.108
C04706=1041.933,326.088,381.281,172.303,42.100,158.109
C04707=1041.941,326.336,381.246,172.307,42.103,158.110
C04708=1041.948,326.584,381.211,172.312,42.105,158.111
C04709=1041.956,326.831,381.176,172.316,42.108,158.112
C04710=1041.963,327.078,381.141,172.321,42.111,158.113
C04711=1041.970,327.326,381.106,172.325,42.113,158.114
C04712=1041.977,327.573,381.071,172.330,42.116,158.115
C04713=1041.984,327.820,381.036,172.335,42.119,158.116
C04714=1041.992,328.068,381.001,172.339,42.122,158.117
C04715=1041.999,328.316,380.966,172.344,42.124,158.118
C04716=1042.007,328.563,380.930,172.348,42.127,158.119
C04717=1042.014,328.810,380.895,172.353,42.130,158.119
C04718=1042.021,329.057,380.860,172.357,42.133,158.120
C04719=1042.028,329.306,380.824,172.362,42.135,158.121
C04720=1042.035,329.552,380.789,172.366,42.138,158.122
C04721=1042.042,329.800,380.753,172.372,42.141,158.123
C04722=1042.050,330.048,380.718,172.376,42.144,158.124
C04723=1042.057,330.294,380.682,172.380,42.147,158.125
C04724=1042.063,330.542,380.647,172.385,42.150,158.126
C04725=1042.071,330.790,380.612,172.389,42.153,158.127
C04726=1042.078,331.037,380.576,172.395,42.156,158.128
C04727=1042.085,331.285,380.540,172.399,42.158,158.129
C04728=1042.092,331.531,380.504,172.404,42.161,158.130
C04729=1042.099,331.779,380.469,172.408,42.164,158.131
C04730=1042.107,332.026,380.433,172.413,42.167,158.132
C04731=1042.114,332.274,380.398,172.417,42.170,158.133
C04732=1042.121,332.521,380.362,172.422,42.173,158.134
C04733=1042.128,332.768,380.326,172.427,42.176,158.135
C04734=1042.136,333.016,380.290,172.432,42.179,158.136
C04735=1042.143,333.263,380.254,172.436,42.182,158.137
C04736=1042.155,333.670,380.195,172.444,42.187,158.139
C04737=1042.167,334.078,380.136,172.452,42.192,158.140
C04738=1042.179,334.486,380.077,172.460,42.197,158.142
C04739=1042.191,334.893,380.019,172.468,42.202,158.144
C04740=1042.198,335.140,379.983,172.472,42.205,158.145
C04741=1042.205,335.388,379.946,172.477,42.208,158.146
C04742=1042.213,335.635,379.910,172.481,42.211,158.147
C04743=1042.220,335.882,379.874,172.487,42.214,158.148
C04744=1042.227,336.130,379.839,172.491,42.217,158.149
C04745=1042.234,336.377,379.802,172.496,42.220,158.150
C04746=1042.241,336.625,379.766,172.500,42.223,158.151
C04747=1042.248,336.871,379.730,172.506,42.226,158.152
C04748=1042.256,337.119,379.694,172.511,42.229,158.153
C04749=1042.263,337.367,379.657,172.515,42.232,158.154
C04750=1042.270,337.613,379.621,172.520,42.235,158.155
C04751=1042.278,337.861,379.585,172.525,42.238,158.156
C04752=1042.284,338.108,379.549,172.530,42.241,158.157
C04753=1042.292,338.355,379.513,172.535,42.244,158.158
C04754=1042.300,338.603,379.476,172.539,42.247,158.159
C04755=1042.307,338.849,379.441,172.545,42.251,158.160
C04756=1042.314,339.097,379.404,172.549,42.254,158.161
C04757=1042.322,339.344,379.367,172.554,42.257,158.162
C04758=1042.329,339.591,379.331,172.559,42.260,158.163
C04759=1042.336,339.838,379.294,172.564,42.264,158.164
C04760=1042.342,340.051,379.263,172.569,42.266,158.165
C04761=1042.348,340.263,379.232,172.573,42.268,158.166
C04762=1042.355,340.476,379.200,172.577,42.271,158.167
C04763=1042.362,340.689,379.169,172.581,42.274,158.168
C04764=1042.368,340.901,379.138,172.585,42.277,158.169
C04765=1042.374,341.114,379.106,172.589,42.280,158.170
C04766=1042.380,341.326,379.075,172.594,42.282,158.171
C04767=1042.387,341.539,379.044,172.598,42.285,158.172
C04768=1042.395,341.786,379.007,172.603,42.288,158.173
C04769=1042.401,342.033,378.970,172.608,42.292,158.174
C04770=1042.409,342.280,378.934,172.613,42.294,158.175
C04771=1042.416,342.527,378.896,172.618,42.298,158.176
C04772=1042.424,342.775,378.860,172.623,42.301,158.177
C04773=1042.431,343.022,378.823,172.628,42.305,158.178
C04774=1042.438,343.269,378.787,172.634,42.308,158.179
C04775=1042.445,343.516,378.749,172.638,42.311,158.181
C04776=1042.453,343.763,378.713,172.643,42.314,158.182
C04777=1042.460,344.010,378.676,172.649,42.318,158.183
C04778=1042.467,344.258,378.639,172.653,42.321,158.184
C04779=1042.475,344.505,378.602,172.658,42.324,158.185
C04780=1042.482,344.752,378.564,172.664,42.328,158.186
C04781=1042.490,344.999,378.528,172.669,42.331,158.187
C04782=1042.497,345.246,378.491,172.673,42.334,158.188
C04783=1042.505,345.493,378.454,172.679,42.338,158.190
C04784=1042.512,345.741,378.417,172.684,42.341,158.191
C04785=1042.519,345.988,378.380,172.690,42.344,158.192
C04786=1042.527,346.235,378.343,172.695,42.348,158.193
C04787=1042.534,346.482,378.306,172.699,42.351,158.194
C04788=1042.541,346.730,378.268,172.705,42.354,158.195
C04789=1042.549,346.976,378.231,172.710,42.358,158.196
C04790=1042.556,347.223,378.194,172.716,42.361,158.198
C04791=1042.564,347.471,378.156,172.721,42.365,158.199
C04792=1042.574,347.806,378.106,172.728,42.369,158.200
C04793=1042.584,348.139,378.056,172.735,42.374,158.202
C04794=1042.594,348.474,378.005,172.742,42.379,158.204
C04795=1042.604,348.808,377.955,172.749,42.383,158.205
C04796=1042.611,349.055,377.918,172.754,42.387,158.206
C04797=1042.619,349.302,377.881,172.759,42.390,158.207
C04798=1042.627,349.550,377.843,172.765,42.394,158.209
C04799=1042.635,349.796,377.805,172.770,42.397,158.210
C04800=1042.643,350.043,377.768,172.776,42.401,158.211
C04801=1042.650,350.290,377.730,172.780,42.404,158.212
C04802=1042.657,350.538,377.693,172.786,42.408,158.213
C04803=1042.664,350.785,377.655,172.791,42.411,158.215
C04804=1042.672,351.032,377.618,172.797,42.415,158.216
C04805=1042.679,351.278,377.579,172.802,42.418,158.217
C04806=1042.687,351.526,377.542,172.808,42.422,158.218
C04807=1042.694,351.773,377.504,172.813,42.425,158.219
C04808=1042.702,352.020,377.467,172.819,42.429,158.221
C04809=1042.710,352.267,377.429,172.824,42.433,158.222
C04810=1042.717,352.514,377.391,172.829,42.437,158.223
C04811=1042.725,352.760,377.353,172.834,42.440,158.224
C04812=1042.732,353.008,377.315,172.839,42.443,158.226
C04813=1042.740,353.255,377.278,172.845,42.448,158.227
C04814=1042.747,353.502,377.239,172.851,42.451,158.228
C04815=1042.754,353.749,377.202,172.856,42.454,158.229
C04816=1042.763,353.996,377.163,172.862,42.459,158.231
C04817=1042.770,354.243,377.126,172.867,42.462,158.232
C04818=1042.777,354.490,377.088,172.873,42.465,158.233
C04819=1042.785,354.737,377.050,172.878,42.470,158.234
C04820=1042.793,354.984,377.011,172.884,42.473,158.236
C04821=1042.800,355.231,376.974,172.889,42.476,158.237
C04822=1042.808,355.478,376.936,172.895,42.481,158.238
C04823=1042.817,355.725,376.898,172.900,42.484,158.239
C04824=1042.824,355.972,376.860,172.906,42.488,158.241
C04825=1042.832,356.219,376.821,172.911,42.491,158.242
C04826=1042.839,356.466,376.783,172.917,42.496,158.243
C04827=1042.847,356.713,376.746,172.923,42.499,158.245
C04828=1042.854,356.960,376.706,172.928,42.503,158.246
C04829=1042.862,357.207,376.668,172.934,42.506,158.247
C04830=1042.869,357.453,376.630,172.939,42.511,158.248
C04831=1042.877,357.700,376.591,172.945,42.514,158.250
C04832=1042.885,357.947,376.553,172.950,42.518,158.251
C04833=1042.893,358.194,376.515,172.956,42.522,158.252
C04834=1042.900,358.441,376.477,172.963,42.525,158.254
C04835=1042.908,358.689,376.438,172.968,42.529,158.255
C04836=1042.915,358.935,376.400,172.974,42.533,158.256
C04837=1042.923,359.183,376.361,172.980,42.537,158.258
C04838=1042.931,359.429,376.323,172.985,42.541,158.259
C04839=1042.939,359.676,376.284,172.991,42.545,158.260
C04840=1042.947,359.922,376.245,172.996,42.549,158.262
C04841=1042.955,360.169,376.207,173.002,42.553,158.263
C04842=1042.962,360.416,376.168,173.008,42.557,158.264
C04843=1042.970,360.664,376.129,173.013,42.560,158.266
C04844=1042.978,360.910,376.091,173.020,42.564,158.267
C04845=1042.986,361.157,376.052,173.026,42.568,158.268
C04846=1042.993,361.403,376.013,173.031,42.572,158.270
C04847=1043.001,361.651,375.974,173.037,42.576,158.271
C04848=1043.012,361.991,375.921,173.045,42.582,158.273
C04849=1043.023,362.331,375.868,173.054,42.587,158.275
C04850=1043.033,362.672,375.814,173.061,42.593,158.277
C04851=1043.045,363.011,375.760,173.069,42.598,158.279
C04852=1043.051,363.258,375.721,173.075,42.603,158.280
C04853=1043.060,363.505,375.682,173.081,42.607,158.282
C04854=1043.067,363.752,375.642,173.088,42.611,158.283
C04855=1043.075,363.998,375.603,173.093,42.615,158.284
C04856=1043.082,364.246,375.564,173.099,42.619,158.286
C04857=1043.091,364.492,375.525,173.105,42.623,158.287
C04858=1043.098,364.739,375.486,173.112,42.627,158.289
C04859=1043.106,364.986,375.447,173.117,42.631,158.290
C04860=1043.114,365.232,375.407,173.123,42.636,158.292
C04861=1043.121,365.479,375.369,173.129,42.640,158.293
C04862=1043.129,365.726,375.329,173.136,42.644,158.294
C04863=1043.138,365.972,375.289,173.141,42.648,158.296
C04864=1043.145,366.219,375.249,173.147,42.652,158.297
C04865=1043.154,366.467,375.211,173.153,42.656,158.299
C04866=1043.161,366.713,375.171,173.160,42.661,158.300
C04867=1043.169,366.959,375.132,173.165,42.665,158.302
C04868=1043.177,367.206,375.092,173.171,42.669,158.303
C04869=1043.185,367.453,375.053,173.178,42.673,158.305
C04870=1043.193,367.700,375.013,173.184,42.678,158.306
C04871=1043.201,367.947,374.974,173.190,42.682,158.307
C04872=1043.208,368.193,374.935,173.197,42.686,158.309
C04873=1043.217,368.440,374.895,173.202,42.690,158.310
C04874=1043.224,368.687,374.855,173.208,42.695,158.312
C04875=1043.233,368.933,374.816,173.215,42.699,158.314
C04876=1043.241,369.180,374.776,173.221,42.703,158.315
C04877=1043.249,369.427,374.737,173.227,42.707,158.316
C04878=1043.257,369.673,374.696,173.234,42.712,158.318
C04879=1043.265,369.920,374.656,173.239,42.716,158.319
C04880=1043.273,370.167,374.617,173.246,42.720,158.321
C04881=1043.281,370.414,374.577,173.252,42.725,158.323
C04882=1043.289,370.660,374.538,173.258,42.729,158.324
C04883=1043.297,370.907,374.498,173.265,42.733,158.325
C04884=1043.305,371.153,374.457,173.271,42.738,158.327
C04885=1043.313,371.400,374.417,173.278,42.742,158.329
C04886=1043.322,371.646,374.377,173.284,42.747,158.330
C04887=1043.329,371.893,374.337,173.291,42.751,158.332
C04888=1043.337,372.140,374.297,173.297,42.756,158.333
C04889=1043.345,372.386,374.257,173.302,42.760,158.335
C04890=1043.353,372.633,374.217,173.309,42.764,158.336
C04891=1043.361,372.879,374.176,173.316,42.770,158.338
C04892=1043.369,373.126,374.136,173.323,42.774,158.340
C04893=1043.377,373.372,374.096,173.328,42.778,158.341
C04894=1043.385,373.619,374.055,173.335,42.783,158.343
C04895=1043.394,373.866,374.015,173.341,42.787,158.344
C04896=1043.402,374.113,373.975,173.348,42.792,158.346
C04897=1043.409,374.359,373.935,173.354,42.797,158.348
C04898=1043.417,374.606,373.894,173.361,42.801,158.349
C04899=1043.426,374.852,373.853,173.367,42.806,158.351
C04900=1043.434,375.098,373.813,173.374,42.810,158.352
C04901=1043.443,375.346,373.773,173.380,42.815,158.354
C04902=1043.451,375.592,373.732,173.387,42.820,158.356
C04903=1043.459,375.838,373.692,173.394,42.824,158.357
C04904=1043.471,376.198,373.633,173.403,42.831,158.360
C04905=1043.483,376.558,373.573,173.413,42.838,158.362
C04906=1043.495,376.918,373.514,173.423,42.845,158.364
C04907=1043.507,377.278,373.455,173.432,42.852,158.367
C04908=1043.515,377.524,373.414,173.439,42.856,158.368
C04909=1043.523,377.771,373.373,173.447,42.861,158.370
C04910=1043.531,378.017,373.333,173.453,42.866,158.372
C04911=1043.540,378.264,373.292,173.460,42.871,158.374
C04912=1043.548,378.510,373.250,173.467,42.875,158.375
C04913=1043.557,378.757,373.209,173.473,42.880,158.377
C04914=1043.566,379.003,373.169,173.480,42.885,158.379
C04915=1043.573,379.250,373.128,173.487,42.890,158.380
C04916=1043.581,379.496,373.087,173.493,42.895,158.382
C04917=1043.590,379.742,373.046,173.500,42.899,158.384
C04918=1043.598,379.989,373.005,173.508,42.904,158.385
C04919=1043.606,380.235,372.963,173.514,42.909,158.387
C04920=1043.614,380.481,372.922,173.521,42.914,158.389
C04921=1043.623,380.728,372.881,173.528,42.919,158.391
C04922=1043.631,380.974,372.840,173.535,42.924,158.392
C04923=1043.640,381.221,372.799,173.541,42.929,158.394
C04924=1043.647,381.467,372.757,173.549,42.934,158.396
C04925=1043.656,381.714,372.716,173.556,42.939,158.398
C04926=1043.664,381.959,372.674,173.563,42.944,158.399
C04927=1043.673,382.206,372.633,173.569,42.949,158.401
C04928=1043.680,382.452,372.592,173.577,42.954,158.403
C04929=1043.689,382.699,372.550,173.584,42.959,158.405
C04930=1043.698,382.945,372.508,173.591,42.964,158.407
C04931=1043.706,383.191,372.467,173.598,42.969,158.408
C04932=1043.714,383.438,372.425,173.605,42.974,158.410
C04933=1043.723,383.684,372.384,173.612,42.979,158.412
C04934=1043.732,383.930,372.342,173.619,42.984,158.414
C04935=1043.740,384.177,372.300,173.626,42.990,158.416
C04936=1043.748,384.423,372.259,173.634,42.994,158.417
C04937=1043.757,384.669,372.217,173.641,42.999,158.419
C04938=1043.766,384.916,372.176,173.648,43.005,158.421
C04939=1043.774,385.162,372.133,173.655,43.010,158.423
C04940=1043.782,385.408,372.092,173.662,43.015,158.425
C04941=1043.791,385.654,372.050,173.669,43.020,158.426
C04942=1043.800,385.901,372.009,173.677,43.026,158.428
C04943=1043.808,386.148,371.966,173.684,43.031,158.430
C04944=1043.817,386.393,371.925,173.691,43.036,158.432
C04945=1043.826,386.639,371.882,173.699,43.041,158.434
C04946=1043.834,386.886,371.840,173.706,43.046,158.436
C04947=1043.843,387.132,371.798,173.713,43.052,158.438
C04948=1043.852,387.378,371.757,173.721,43.057,158.440
C04949=1043.860,387.625,371.714,173.728,43.062,158.442
C04950=1043.869,387.871,371.672,173.735,43.067,158.443
C04951=1043.878,388.117,371.630,173.743,43.073,158.445
C04952=1043.887,388.363,371.589,173.750,43.078,158.447
C04953=1043.895,388.609,371.546,173.758,43.083,158.449
C04954=1043.904,388.855,371.504,173.765,43.089,158.451
C04955=1043.912,389.102,371.462,173.773,43.094,158.453
C04956=1043.921,389.348,371.419,173.780,43.100,158.455
C04957=1043.930,389.594,371.376,173.788,43.105,158.457
C04958=1043.938,389.840,371.334,173.795,43.110,158.459
C04959=1043.948,390.086,371.292,173.803,43.116,158.461
C04960=1043.961,390.480,371.223,173.815,43.125,158.464
C04961=1043.975,390.873,371.155,173.828,43.133,158.467
C04962=1043.989,391.266,371.088,173.840,43.142,158.470
C04963=1044.003,391.661,371.019,173.852,43.151,158.473
C04964=1044.012,391.907,370.976,173.859,43.157,158.476
C04965=1044.021,392.152,370.934,173.867,43.162,158.477
C04966=1044.030,392.399,370.891,173.875,43.168,158.480
C04967=1044.038,392.645,370.848,173.883,43.174,158.482
C04968=1044.047,392.890,370.805,173.891,43.179,158.484
C04969=1044.056,393.136,370.762,173.898,43.185,158.486
C04970=1044.064,393.382,370.719,173.906,43.191,158.488
C04971=1044.073,393.629,370.676,173.914,43.197,158.490
C04972=1044.083,393.875,370.633,173.922,43.202,158.492
C04973=1044.091,394.120,370.590,173.930,43.208,158.494
C04974=1044.100,394.366,370.547,173.937,43.214,158.496
C04975=1044.109,394.613,370.503,173.945,43.220,158.498
C04976=1044.118,394.859,370.461,173.954,43.225,158.500
C04977=1044.127,395.104,370.417,173.961,43.231,158.502
C04978=1044.136,395.350,370.374,173.969,43.237,158.504
C04979=1044.145,395.597,370.331,173.978,43.242,158.507
C04980=1044.154,395.842,370.288,173.986,43.248,158.509
C04981=1044.163,396.088,370.245,173.993,43.254,158.511
C04982=1044.172,396.334,370.200,174.002,43.260,158.513
C04983=1044.181,396.580,370.157,174.010,43.266,158.515
C04984=1044.189,396.826,370.114,174.018,43.272,158.517
C04985=1044.199,397.073,370.070,174.026,43.278,158.519
C04986=1044.207,397.318,370.027,174.034,43.284,158.522
C04987=1044.216,397.565,369.983,174.042,43.290,158.524
C04988=1044.225,397.810,369.939,174.051,43.296,158.526
C04989=1044.235,398.056,369.895,174.059,43.302,158.528
C04990=1044.244,398.302,369.852,174.067,43.308,158.530
C04991=1044.253,398.549,369.808,174.075,43.314,158.533
C04992=1044.261,398.794,369.764,174.083,43.320,158.535
C04993=1044.271,399.040,369.720,174.092,43.326,158.537
C04994=1044.280,399.286,369.677,174.100,43.332,158.539
C04995=1044.289,399.532,369.632,174.109,43.339,158.541
C04996=1044.298,399.778,369.588,174.116,43.344,158.544
C04997=1044.307,400.023,369.545,174.125,43.351,158.546
C04998=1044.317,400.269,369.500,174.133,43.357,158.548
C04999=1044.326,400.516,369.456,174.142,43.363,158.550
C05000=1044.335,400.761,369.413,174.150,43.369,158.553
C05001=1044.344,401.007,369.369,174.159,43.375,158.555
C05002=1044.354,401.253,369.324,174.168,43.381,158.557
C05003=1044.363,401.499,369.281,174.176,43.388,158.560
C05004=1044.372,401.744,369.236,174.185,43.394,158.562
C05005=1044.382,401.990,369.192,174.193,43.400,158.564
C05006=1044.390,402.237,369.147,174.202,43.406,158.566
C05007=1044.399,402.482,369.103,174.211,43.413,158.569
C05008=1044.409,402.728,369.058,174.219,43.419,158.571
C05009=1044.418,402.974,369.014,174.228,43.426,158.574
C05010=1044.428,403.219,368.970,174.236,43.432,158.576
C05011=1044.437,403.466,368.925,174.245,43.438,158.578
C05012=1044.446,403.711,368.880,174.254,43.445,158.581
C05013=1044.456,403.958,368.836,174.262,43.451,158.583
C05014=1044.464,404.203,368.791,174.271,43.458,158.585
C05015=1044.474,404.448,368.746,174.280,43.464,158.588
C05016=1044.490,404.861,368.671,174.295,43.475,158.592
C05017=1044.505,405.274,368.596,174.310,43.486,158.596
C05018=1044.520,405.686,368.520,174.325,43.497,158.600
C05019=1044.537,406.099,368.445,174.340,43.509,158.604
C05020=1044.546,406.345,368.399,174.349,43.515,158.607
C05021=1044.555,406.590,368.355,174.358,43.522,158.609
C05022=1044.565,406.836,368.310,174.367,43.528,158.612
C05023=1044.575,407.082,368.264,174.377,43.535,158.614
C05024=1044.584,407.328,368.219,174.386,43.542,158.617
C05025=1044.593,407.574,368.174,174.395,43.549,158.619
C05026=1044.603,407.818,368.128,174.403,43.555,158.622
C05027=1044.612,408.064,368.083,174.413,43.562,158.624
C05028=1044.623,408.311,368.038,174.422,43.569,158.627
C05029=1044.632,408.556,367.992,174.431,43.576,158.629
C05030=1044.642,408.801,367.947,174.441,43.582,158.632
C05031=1044.651,409.047,367.901,174.450,43.589,158.634
C05032=1044.661,409.293,367.856,174.459,43.596,158.637
C05033=1044.671,409.538,367.810,174.469,43.603,158.640
C05034=1044.680,409.784,367.765,174.478,43.610,158.642
C05035=1044.691,410.030,367.719,174.487,43.616,158.645
C05036=1044.700,410.275,367.674,174.497,43.624,158.647
C05037=1044.710,410.521,367.628,174.506,43.630,158.650
C05038=1044.719,410.767,367.582,174.516,43.638,158.653
C05039=1044.729,411.012,367.537,174.526,43.644,158.655
C05040=1044.739,411.258,367.491,174.535,43.651,158.658
C05041=1044.749,411.504,367.445,174.545,43.658,158.661
C05042=1044.759,411.749,367.399,174.554,43.665,158.663
C05043=1044.769,411.995,367.353,174.564,43.672,158.666
C05044=1044.778,412.240,367.308,174.573,43.680,158.669
C05045=1044.788,412.486,367.261,174.583,43.687,158.671
C05046=1044.798,412.731,367.216,174.594,43.694,158.674
C05047=1044.808,412.977,367.169,174.603,43.701,158.677
C05048=1044.817,413.222,367.123,174.613,43.708,158.679
C05049=1044.827,413.468,367.076,174.622,43.715,158.682
C05050=1044.837,413.714,367.029,174.632,43.723,158.685
C05051=1044.847,413.958,366.984,174.642,43.730,158.688
C05052=1044.857,414.204,366.937,174.652,43.737,158.690
C05053=1044.867,414.450,366.891,174.662,43.745,158.693
C05054=1044.877,414.695,366.844,174.672,43.752,158.696
C05055=1044.887,414.941,366.797,174.682,43.759,158.699
C05056=1044.897,415.187,366.751,174.692,43.766,158.702
C05057=1044.907,415.432,366.704,174.703,43.774,158.704
C05058=1044.917,415.678,366.658,174.712,43.781,158.707
C05059=1044.927,415.922,366.611,174.722,43.789,158.710
C05060=1044.937,416.168,366.564,174.733,43.796,158.713
C05061=1044.947,416.413,366.517,174.742,43.804,158.716
C05062=1044.957,416.659,366.471,174.753,43.811,158.719
C05063=1044.968,416.904,366.424,174.763,43.819,158.722
C05064=1044.978,417.149,366.377,174.774,43.826,158.725
C05065=1044.988,417.395,366.330,174.784,43.834,158.727
C05066=1044.998,417.641,366.283,174.795,43.842,158.730
C05067=1045.008,417.886,366.236,174.805,43.849,158.733
C05068=1045.018,418.131,366.189,174.815,43.857,158.736
C05069=1045.029,418.377,366.141,174.826,43.864,158.739
C05070=1045.039,418.622,366.094,174.836,43.872,158.742
C05071=1045.049,418.867,366.047,174.847,43.879,158.745
C05072=1045.058,419.078,366.007,174.855,43.886,158.748
C05073=1045.067,419.288,365.966,174.865,43.893,158.750
C05074=1045.075,419.498,365.926,174.874,43.899,158.753
C05075=1045.084,419.708,365.885,174.883,43.907,158.755
C05076=1045.093,419.918,365.844,174.892,43.913,158.758
C05077=1045.102,420.129,365.803,174.902,43.920,158.761
C05078=1045.111,420.338,365.763,174.911,43.926,158.763
C05079=1045.120,420.548,365.722,174.920,43.933,158.766
C05080=1045.130,420.794,365.675,174.931,43.941,158.769
C05081=1045.141,421.039,365.627,174.942,43.949,158.772
C05082=1045.150,421.285,365.579,174.953,43.957,158.775
C05083=1045.161,421.529,365.531,174.964,43.965,158.778
C05084=1045.171,421.775,365.484,174.974,43.973,158.781
C05085=1045.182,422.020,365.435,174.985,43.981,158.785
C05086=1045.193,422.265,365.388,174.997,43.989,158.788
C05087=1045.203,422.510,365.340,175.008,43.997,158.791
C05088=1045.214,422.755,365.292,175.019,44.005,158.794
C05089=1045.224,423.000,365.244,175.030,44.013,158.797
C05090=1045.235,423.246,365.195,175.041,44.021,158.800
C05091=1045.245,423.491,365.148,175.053,44.029,158.804
C05092=1045.256,423.736,365.100,175.064,44.037,158.807
C05093=1045.266,423.981,365.052,175.075,44.046,158.810
C05094=1045.278,424.226,365.003,175.086,44.054,158.813
C05095=1045.287,424.471,364.955,175.098,44.062,158.817
C05096=1045.298,424.717,364.907,175.109,44.070,158.820
C05097=1045.310,424.962,364.858,175.120,44.078,158.823
C05098=1045.320,425.206,364.810,175.132,44.087,158.826
C05099=1045.331,425.452,364.761,175.143,44.095,158.830
C05100=1045.341,425.696,364.713,175.155,44.104,158.833
C05101=1045.352,425.941,364.663,175.166,44.112,158.836
C05102=1045.363,426.187,364.615,175.179,44.120,158.840
C05103=1045.374,426.431,364.566,175.190,44.129,158.843
C05104=1045.384,426.677,364.517,175.202,44.137,158.846
C05105=1045.396,426.921,364.468,175.213,44.146,158.850
C05106=1045.406,427.167,364.420,175.226,44.154,158.853
C05107=1045.417,427.411,364.371,175.237,44.163,158.857
C05108=1045.428,427.656,364.322,175.249,44.171,158.860
C05109=1045.438,427.901,364.273,175.261,44.180,158.863
C05110=1045.450,428.146,364.224,175.273,44.188,158.867
C05111=1045.461,428.391,364.174,175.285,44.197,158.870
C05112=1045.472,428.636,364.125,175.298,44.206,158.874
C05113=1045.483,428.881,364.076,175.309,44.214,158.877
C05114=1045.494,429.126,364.027,175.321,44.223,158.881
C05115=1045.505,429.371,363.977,175.334,44.232,158.884
C05116=1045.515,429.616,363.928,175.345,44.241,158.888
C05117=1045.527,429.861,363.878,175.358,44.250,158.891
C05118=1045.537,430.106,363.829,175.370,44.259,158.895
C05119=1045.549,430.350,363.779,175.383,44.268,158.899
C05120=1045.560,430.595,363.730,175.395,44.277,158.902
C05121=1045.570,430.840,363.680,175.407,44.285,158.906
C05122=1045.582,431.084,363.630,175.420,44.295,158.910
C05123=1045.593,431.329,363.581,175.432,44.303,158.913
C05124=1045.604,431.573,363.530,175.445,44.313,158.917
C05125=1045.616,431.819,363.481,175.458,44.321,158.921
C05126=1045.627,432.063,363.431,175.470,44.331,158.924
C05127=1045.638,432.308,363.380,175.483,44.340,158.928
C05128=1045.649,432.552,363.331,175.496,44.348,158.932
C05129=1045.661,432.798,363.281,175.509,44.358,158.935
C05130=1045.672,433.042,363.230,175.521,44.367,158.939
C05131=1045.683,433.286,363.180,175.534,44.376,158.943
C05132=1045.698,433.610,363.114,175.552,44.388,158.948
C05133=1045.714,433.933,363.047,175.569,44.400,158.953
C05134=1045.729,434.255,362.981,175.587,44.413,158.958
C05135=1045.744,434.578,362.915,175.604,44.425,158.963
C05136=1045.756,434.822,362.864,175.617,44.434,158.967
C05137=1045.767,435.067,362.813,175.630,44.444,158.971
C05138=1045.779,435.312,362.763,175.643,44.453,158.975
C05139=1045.790,435.555,362.712,175.657,44.463,158.979
C05140=1045.802,435.801,362.661,175.670,44.472,158.983
C05141=1045.814,436.046,362.611,175.684,44.482,158.987
C05142=1045.825,436.290,362.560,175.698,44.491,158.990
C05143=1045.837,436.534,362.509,175.711,44.501,158.994
C05144=1045.849,436.779,362.458,175.724,44.510,158.998
C05145=1045.860,437.023,362.407,175.738,44.520,159.002
C05146=1045.872,437.267,362.356,175.751,44.530,159.006
C05147=1045.884,437.512,362.304,175.766,44.540,159.011
C05148=1045.896,437.756,362.253,175.779,44.549,159.015
C05149=1045.908,438.001,362.202,175.793,44.559,159.019
C05150=1045.919,438.246,362.151,175.808,44.569,159.023
C05151=1045.932,438.490,362.099,175.821,44.579,159.027
C05152=1045.943,438.734,362.048,175.836,44.588,159.031
C05153=1045.955,438.978,361.996,175.849,44.598,159.035
C05154=1045.967,439.223,361.945,175.863,44.608,159.039
C05155=1045.979,439.467,361.894,175.878,44.618,159.044
C05156=1045.991,439.711,361.841,175.892,44.628,159.048
C05157=1046.003,439.955,361.790,175.906,44.638,159.052
C05158=1046.015,440.199,361.738,175.921,44.648,159.056
C05159=1046.027,440.445,361.686,175.935,44.658,159.060
C05160=1046.039,440.688,361.634,175.950,44.668,159.065
C05161=1046.051,440.933,361.583,175.965,44.678,159.069
C05162=1046.064,441.177,361.530,175.978,44.688,159.073
C05163=1046.076,441.422,361.477,175.993,44.699,159.078
C05164=1046.088,441.666,361.425,176.009,44.709,159.082
C05165=1046.100,441.910,361.373,176.023,44.719,159.087
C05166=1046.112,442.153,361.321,176.037,44.729,159.091
C05167=1046.125,442.398,361.269,176.052,44.739,159.095
C05168=1046.137,442.642,361.216,176.068,44.750,159.100
C05169=1046.149,442.886,361.164,176.083,44.760,159.104
C05170=1046.161,443.131,361.111,176.098,44.771,159.109
C05171=1046.174,443.375,361.059,176.113,44.781,159.113
C05172=1046.192,443.738,360.980,176.135,44.797,159.120
C05173=1046.211,444.101,360.902,176.158,44.812,159.127
C05174=1046.229,444.464,360.824,176.181,44.828,159.133
C05175=1046.249,444.827,360.745,176.204,44.844,159.140
C05176=1046.261,445.071,360.692,176.220,44.854,159.145
C05177=1046.273,445.314,360.640,176.235,44.865,159.150
C05178=1046.286,445.557,360.587,176.251,44.876,159.154
C05179=1046.300,445.801,360.534,176.267,44.886,159.159
C05180=1046.314,446.043,360.482,176.282,44.897,159.163
C05181=1046.328,446.287,360.431,176.298,44.907,159.168
C05182=1046.344,446.532,360.380,176.315,44.917,159.173
C05183=1046.359,446.775,360.330,176.331,44.927,159.177
C05184=1046.377,447.019,360.280,176.347,44.937,159.182
C05185=1046.394,447.263,360.230,176.363,44.947,159.186
C05186=1046.412,447.507,360.182,176.379,44.956,159.190
C05187=1046.431,447.752,360.133,176.395,44.966,159.195
C05188=1046.454,448.052,360.075,176.415,44.978,159.200
C05189=1046.479,448.352,360.017,176.436,44.989,159.206
C05190=1046.505,448.654,359.960,176.456,45.000,159.211
C05191=1046.531,448.955,359.903,176.477,45.011,159.216
C05192=1046.554,449.200,359.858,176.494,45.020,159.221
C05193=1046.577,449.445,359.813,176.511,45.028,159.225
C05194=1046.601,449.690,359.768,176.527,45.037,159.229
C05195=1046.625,449.935,359.725,176.545,45.045,159.233
C05196=1046.650,450.181,359.682,176.562,45.054,159.238
C05197=1046.676,450.426,359.639,176.579,45.062,159.242
C05198=1046.703,450.672,359.597,176.596,45.069,159.246
C05199=1046.730,450.916,359.555,176.613,45.078,159.250
C05200=1046.422,450.951,359.248,176.615,45.163,159.275
C05201=1046.395,450.706,359.289,176.598,45.155,159.271
C05202=1046.368,450.461,359.332,176.580,45.147,159.267
C05203=1046.343,450.215,359.374,176.563,45.139,159.263
C05204=1046.317,449.971,359.417,176.546,45.131,159.259
C05205=1046.292,449.725,359.461,176.528,45.123,159.254
C05206=1046.268,449.480,359.505,176.512,45.114,159.250
C05207=1046.246,449.235,359.549,176.495,45.105,159.246
C05208=1046.223,448.990,359.595,176.478,45.097,159.242
C05209=1046.197,448.706,359.648,176.458,45.087,159.237
C05210=1046.173,448.421,359.702,176.438,45.076,159.232
C05211=1046.149,448.138,359.757,176.420,45.066,159.227
C05212=1046.126,447.854,359.812,176.401,45.055,159.222
C05213=1046.107,447.609,359.860,176.383,45.046,159.217
C05214=1046.089,447.366,359.908,176.368,45.037,159.213
C05215=1046.071,447.121,359.957,176.351,45.027,159.208
C05216=1046.055,446.878,360.007,176.335,45.017,159.204
C05217=1046.038,446.634,360.057,176.319,45.007,159.199
C05218=1046.022,446.390,360.108,176.303,44.997,159.195
C05219=1046.007,446.146,360.158,176.287,44.987,159.190
C05220=1045.992,445.903,360.210,176.270,44.977,159.185
C05221=1045.979,445.658,360.262,176.255,44.966,159.181
C05222=1045.966,445.415,360.315,176.240,44.956,159.176
C05223=1045.953,445.173,360.368,176.223,44.946,159.172
C05224=1045.940,444.930,360.421,176.208,44.935,159.167
C05225=1045.928,444.686,360.473,176.192,44.924,159.162
C05226=1045.915,444.442,360.526,176.177,44.914,159.158
C05227=1045.902,444.198,360.579,176.162,44.903,159.153
C05228=1045.890,443.954,360.632,176.145,44.893,159.149
C05229=1045.877,443.710,360.685,176.130,44.883,159.144
C05230=1045.865,443.466,360.738,176.115,44.872,159.139
C05231=1045.852,443.221,360.790,176.100,44.862,159.135
C05232=1045.840,442.977,360.842,176.085,44.852,159.131
C05233=1045.827,442.733,360.895,176.070,44.841,159.126
C05234=1045.815,442.489,360.947,176.054,44.831,159.122
C05235=1045.803,442.245,361.000,176.039,44.821,159.117
C05236=1045.791,442.001,361.053,176.025,44.810,159.113
C05237=1045.779,441.757,361.105,176.010,44.800,159.108
C05238=1045.766,441.513,361.157,175.995,44.790,159.104
C05239=1045.754,441.269,361.209,175.980,44.780,159.100
C05240=1045.742,441.024,361.261,175.965,44.770,159.095
C05241=1045.729,440.780,361.313,175.951,44.760,159.091
C05242=1045.717,440.536,361.365,175.936,44.749,159.087
C05243=1045.705,440.291,361.416,175.922,44.740,159.082
C05244=1045.693,440.047,361.469,175.908,44.730,159.078
C05245=1045.681,439.803,361.520,175.893,44.720,159.074
C05246=1045.669,439.558,361.572,175.878,44.710,159.070
C05247=1045.657,439.314,361.624,175.865,44.700,159.066
C05248=1045.645,439.069,361.675,175.850,44.690,159.061
C05249=1045.633,438.825,361.727,175.836,44.680,159.057
C05250=1045.621,438.582,361.778,175.822,44.671,159.053
C05251=1045.609,438.337,361.830,175.808,44.661,159.049
C05252=1045.598,438.093,361.881,175.794,44.651,159.045
C05253=1045.582,437.778,361.948,175.776,44.639,159.039
C05254=1045.567,437.463,362.014,175.758,44.626,159.034
C05255=1045.552,437.148,362.079,175.740,44.614,159.029
C05256=1045.537,436.833,362.145,175.723,44.601,159.024
C05257=1045.526,436.589,362.196,175.708,44.592,159.020
C05258=1045.514,436.344,362.248,175.695,44.583,159.016
C05259=1045.502,436.099,362.298,175.681,44.573,159.012
C05260=1045.489,435.855,362.349,175.668,44.563,159.008
C05261=1045.478,435.611,362.400,175.655,44.554,159.004
C05262=1045.467,435.366,362.451,175.641,44.545,159.000
C05263=1045.455,435.121,362.502,175.628,44.535,158.996
C05264=1045.443,434.877,362.551,175.614,44.526,158.992
C05265=1045.425,434.504,362.629,175.594,44.512,158.986
C05266=1045.408,434.130,362.707,175.574,44.498,158.980
C05267=1045.389,433.756,362.783,175.554,44.484,158.975
C05268=1045.373,433.383,362.860,175.534,44.469,158.969
C05269=1045.362,433.138,362.910,175.521,44.460,158.965
C05270=1045.350,432.893,362.960,175.508,44.452,158.961
C05271=1045.339,432.648,363.010,175.495,44.442,158.958
C05272=1045.327,432.403,363.061,175.482,44.433,158.954
C05273=1045.315,432.159,363.110,175.470,44.424,158.950
C05274=1045.305,431.914,363.160,175.457,44.415,158.946
C05275=1045.294,431.670,363.210,175.444,44.406,158.943
C05276=1045.281,431.425,363.260,175.431,44.398,158.939
C05277=1045.271,431.180,363.310,175.419,44.388,158.935
C05278=1045.260,430.935,363.360,175.406,44.379,158.932
C05279=1045.248,430.691,363.409,175.393,44.371,158.928
C05280=1045.237,430.446,363.460,175.381,44.361,158.924
C05281=1045.227,430.201,363.509,175.368,44.353,158.921
C05282=1045.215,429.956,363.558,175.356,44.344,158.917
C05283=1045.205,429.711,363.608,175.344,44.335,158.914
C05284=1045.194,429.467,363.658,175.332,44.326,158.910
C05285=1045.182,429.222,363.707,175.319,44.318,158.907
C05286=1045.172,428.977,363.757,175.307,44.309,158.903
C05287=1045.160,428.732,363.806,175.295,44.301,158.900
C05288=1045.149,428.487,363.856,175.283,44.292,158.896
C05289=1045.138,428.243,363.905,175.270,44.283,158.893
C05290=1045.127,427.998,363.954,175.259,44.275,158.889
C05291=1045.116,427.752,364.002,175.246,44.266,158.886
C05292=1045.106,427.507,364.052,175.234,44.257,158.882
C05293=1045.094,427.262,364.101,175.223,44.249,158.879
C05294=1045.084,427.018,364.149,175.210,44.241,158.875
C05295=1045.073,426.773,364.199,175.199,44.232,158.872
C05296=1045.062,426.528,364.248,175.187,44.223,158.869
C05297=1045.051,426.283,364.296,175.175,44.215,158.865
C05298=1045.040,426.038,364.345,175.163,44.207,158.862
C05299=1045.029,425.793,364.393,175.151,44.198,158.858
C05300=1045.019,425.547,364.442,175.140,44.191,158.855
C05301=1045.008,425.303,364.491,175.129,44.182,158.852
C05302=1044.997,425.058,364.539,175.117,44.174,158.849
C05303=1044.987,424.812,364.588,175.106,44.165,158.845
C05304=1044.976,424.567,364.636,175.095,44.157,158.842
C05305=1044.965,424.322,364.684,175.082,44.149,158.839
C05306=1044.955,424.077,364.732,175.071,44.141,158.836
C05307=1044.944,423.832,364.781,175.059,44.133,158.832
C05308=1044.933,423.586,364.830,175.048,44.125,158.829
C05309=1044.923,423.342,364.877,175.037,44.117,158.826
C05310=1044.912,423.096,364.926,175.025,44.108,158.823
C05311=1044.901,422.852,364.974,175.014,44.100,158.819
C05312=1044.891,422.607,365.022,175.003,44.092,158.816
C05313=1044.880,422.361,365.069,174.992,44.085,158.813
C05314=1044.869,422.116,365.117,174.982,44.076,158.810
C05315=1044.859,421.871,365.166,174.970,44.068,158.807
C05316=1044.849,421.625,365.213,174.959,44.060,158.804
C05317=1044.838,421.381,365.261,174.948,44.052,158.801
C05318=1044.827,421.135,365.309,174.937,44.045,158.798
C05319=1044.817,420.890,365.357,174.926,44.037,158.794
C05320=1044.807,420.645,365.404,174.916,44.029,158.791
C05321=1044.798,420.434,365.446,174.906,44.022,158.789
C05322=1044.789,420.223,365.486,174.897,44.016,158.786
C05323=1044.780,420.011,365.527,174.887,44.009,158.783
C05324=1044.771,419.800,365.568,174.878,44.002,158.781
C05325=1044.763,419.589,365.609,174.869,43.995,158.778
C05326=1044.754,419.378,365.650,174.860,43.989,158.776
C05327=1044.745,419.166,365.691,174.851,43.982,158.773
C05328=1044.736,418.955,365.731,174.841,43.976,158.770
C05329=1044.726,418.710,365.779,174.831,43.968,158.767
C05330=1044.716,418.465,365.826,174.820,43.960,158.764
C05331=1044.705,418.219,365.874,174.809,43.953,158.761
C05332=1044.695,417.974,365.921,174.799,43.945,158.758
C05333=1044.684,417.728,365.968,174.788,43.938,158.755
C05334=1044.675,417.482,366.014,174.778,43.930,158.753
C05335=1044.664,417.237,366.062,174.768,43.923,158.750
C05336=1044.654,416.992,366.109,174.758,43.915,158.747
C05337=1044.643,416.747,366.155,174.747,43.908,158.744
C05338=1044.633,416.501,366.202,174.737,43.900,158.741
C05339=1044.624,416.256,366.249,174.727,43.893,158.738
C05340=1044.614,416.010,366.295,174.717,43.885,158.735
C05341=1044.604,415.765,366.343,174.706,43.878,158.733
C05342=1044.593,415.520,366.389,174.696,43.871,158.730
C05343=1044.583,415.274,366.436,174.686,43.864,158.727
C05344=1044.573,415.028,366.482,174.676,43.856,158.724
C05345=1044.563,414.784,366.529,174.666,43.849,158.721
C05346=1044.554,414.538,366.576,174.655,43.841,158.718
C05347=1044.544,414.292,366.622,174.646,43.834,158.716
C05348=1044.533,414.047,366.669,174.636,43.827,158.713
C05349=1044.523,413.802,366.715,174.625,43.820,158.710
C05350=1044.514,413.556,366.761,174.616,43.813,158.707
C05351=1044.504,413.311,366.807,174.606,43.806,158.705
C05352=1044.494,413.065,366.854,174.596,43.799,158.702
C05353=1044.484,412.819,366.900,174.586,43.791,158.699
C05354=1044.474,412.574,366.946,174.576,43.784,158.696
C05355=1044.465,412.328,366.992,174.567,43.777,158.694
C05356=1044.455,412.083,367.039,174.557,43.770,158.691
C05357=1044.445,411.837,367.085,174.547,43.763,158.688
C05358=1044.435,411.591,367.131,174.537,43.756,158.686
C05359=1044.425,411.346,367.177,174.528,43.749,158.683
C05360=1044.414,411.100,367.222,174.518,43.742,158.680
C05361=1044.405,410.855,367.268,174.509,43.735,158.678
C05362=1044.395,410.609,367.314,174.499,43.728,158.675
C05363=1044.386,410.364,367.359,174.490,43.721,158.672
C05364=1044.376,410.119,367.405,174.480,43.715,158.670
C05365=1044.366,409.872,367.451,174.470,43.707,158.667
C05366=1044.356,409.627,367.496,174.461,43.701,158.664
C05367=1044.346,409.381,367.542,174.451,43.694,158.662
C05368=1044.336,409.136,367.587,174.442,43.687,158.659
C05369=1044.327,408.890,367.633,174.433,43.681,158.657
C05370=1044.317,408.644,367.678,174.423,43.673,158.654
C05371=1044.308,408.399,367.724,174.414,43.667,158.652
C05372=1044.298,408.153,367.769,174.404,43.660,158.649
C05373=1044.289,407.907,367.814,174.395,43.653,158.647
C05374=1044.279,407.661,367.860,174.386,43.647,158.644
C05375=1044.269,407.416,367.904,174.378,43.640,158.641
C05376=1044.260,407.170,367.950,174.368,43.633,158.639
C05377=1044.250,406.925,367.995,174.359,43.627,158.637
C05378=1044.241,406.679,368.041,174.350,43.620,158.634
C05379=1044.231,406.434,368.086,174.341,43.613,158.632
C05380=1044.222,406.188,368.131,174.332,43.607,158.629
C05381=1044.206,405.773,368.207,174.316,43.596,158.625
C05382=1044.190,405.359,368.282,174.302,43.585,158.621
C05383=1044.174,404.943,368.359,174.286,43.574,158.617
C05384=1044.159,404.529,368.434,174.271,43.563,158.613
C05385=1044.150,404.283,368.479,174.262,43.557,158.610
C05386=1044.140,404.037,368.524,174.254,43.550,158.608
C05387=1044.131,403.791,368.568,174.245,43.543,158.605
C05388=1044.121,403.546,368.613,174.236,43.537,158.603
C05389=1044.112,403.299,368.658,174.228,43.531,158.601
C05390=1044.103,403.054,368.702,174.218,43.525,158.598
C05391=1044.093,402.807,368.747,174.209,43.518,158.596
C05392=1044.084,402.563,368.791,174.201,43.512,158.594
C05393=1044.075,402.316,368.836,174.192,43.506,158.591
C05394=1044.066,402.071,368.881,174.183,43.500,158.589
C05395=1044.056,401.825,368.925,174.175,43.493,158.587
C05396=1044.047,401.578,368.969,174.166,43.487,158.584
C05397=1044.038,401.333,369.013,174.157,43.481,158.582
C05398=1044.028,401.087,369.057,174.149,43.474,158.580
C05399=1044.019,400.841,369.101,174.141,43.469,158.577
C05400=1044.010,400.596,369.145,174.132,43.462,158.575
C05401=1044.002,400.349,369.190,174.123,43.456,158.573
C05402=1043.992,400.103,369.234,174.116,43.450,158.571
C05403=1043.983,399.857,369.278,174.107,43.444,158.568
C05404=1043.974,399.612,369.322,174.099,43.437,158.566
C05405=1043.964,399.366,369.366,174.090,43.432,158.564
C05406=1043.955,399.121,369.409,174.082,43.426,158.562
C05407=1043.946,398.874,369.453,174.073,43.420,158.559
C05408=1043.937,398.628,369.496,174.065,43.414,158.557
C05409=1043.928,398.382,369.540,174.056,43.408,158.555
C05410=1043.918,398.136,369.584,174.049,43.402,158.553
C05411=1043.909,397.891,369.628,174.040,43.396,158.551
C05412=1043.900,397.644,369.672,174.032,43.390,158.548
C05413=1043.891,397.398,369.715,174.023,43.384,158.546
C05414=1043.883,397.153,369.759,174.015,43.378,158.544
C05415=1043.874,396.906,369.802,174.008,43.372,158.542
C05416=1043.865,396.661,369.846,173.999,43.366,158.540
C05417=1043.855,396.415,369.890,173.991,43.360,158.538
C05418=1043.847,396.169,369.933,173.982,43.355,158.535
C05419=1043.838,395.923,369.977,173.975,43.349,158.533
C05420=1043.829,395.676,370.020,173.967,43.343,158.531
C05421=1043.820,395.431,370.063,173.958,43.337,158.529
C05422=1043.811,395.185,370.107,173.950,43.331,158.527
C05423=1043.802,394.938,370.150,173.943,43.325,158.525
C05424=1043.793,394.692,370.193,173.934,43.320,158.523
C05425=1043.784,394.447,370.236,173.926,43.314,158.521
C05426=1043.775,394.201,370.279,173.919,43.308,158.519
C05427=1043.766,393.955,370.323,173.911,43.303,158.517
C05428=1043.757,393.709,370.365,173.902,43.297,158.514
C05429=1043.748,393.463,370.408,173.895,43.291,158.512
C05430=1043.740,393.217,370.451,173.887,43.286,158.510
C05431=1043.730,392.971,370.495,173.879,43.280,158.508
C05432=1043.721,392.725,370.538,173.871,43.275,158.506
C05433=1043.713,392.479,370.581,173.863,43.269,158.504
C05434=1043.704,392.233,370.624,173.856,43.264,158.502
C05435=1043.696,391.987,370.667,173.848,43.258,158.500
C05436=1043.687,391.740,370.708,173.840,43.252,158.498
C05437=1043.673,391.345,370.778,173.827,43.244,158.495
C05438=1043.659,390.950,370.846,173.815,43.235,158.492
C05439=1043.645,390.554,370.914,173.803,43.226,158.489
C05440=1043.631,390.159,370.983,173.791,43.217,158.485
C05441=1043.622,389.913,371.026,173.784,43.212,158.483
C05442=1043.613,389.666,371.067,173.775,43.206,158.481
C05443=1043.605,389.420,371.110,173.768,43.201,158.479
C05444=1043.595,389.174,371.153,173.760,43.196,158.478
C05445=1043.587,388.928,371.195,173.753,43.190,158.476
C05446=1043.578,388.682,371.238,173.745,43.185,158.474
C05447=1043.570,388.435,371.280,173.738,43.179,158.472
C05448=1043.561,388.189,371.322,173.730,43.174,158.470
C05449=1043.552,387.943,371.365,173.723,43.169,158.468
C05450=1043.543,387.696,371.406,173.716,43.164,158.466
C05451=1043.534,387.450,371.448,173.708,43.158,158.464
C05452=1043.526,387.204,371.490,173.701,43.153,158.462
C05453=1043.517,386.958,371.533,173.693,43.148,158.460
C05454=1043.509,386.712,371.574,173.686,43.143,158.458
C05455=1043.500,386.466,371.616,173.679,43.137,158.457
C05456=1043.492,386.219,371.658,173.671,43.133,158.455
C05457=1043.483,385.973,371.700,173.664,43.127,158.453
